// TIA Portal V16 program export: 7 tag tables, 0 data types, 4 data blocks, 31 code blocks (in call order from the OBs), 28 instance data blocks

VAR_GLOBAL   // PLC tag table "100固定地址变量表"
   ManAutoPB AT %I1.0 : Bool;   // 手动/自动   {ExternalVisible false}
   StartPB AT %I1.1 : Bool;   // 启动(固定)
   StopPB AT %I1.2 : Bool;   // 停止(固定)
   RestPB AT %I1.3 : Bool;   // 复位(固定)
   EM_PB AT %I1.4 : Bool;   // 急停(固定)
   Buzzer AT %Q0.4 : Bool;   // 蜂鸣器Bz
   R_LED AT %Q0.5 : Bool;   // 三色灯<红>
   G_LED AT %Q0.6 : Bool;   // 三色灯<绿>
   Y_LED AT %Q0.7 : Bool;   // 三色灯<黄>
   Auto_LED AT %Q1.0 : Bool;   // 自动灯
   Clock_Byte AT %MB0 : Byte;
   System_Byte AT %MB1 : Byte;
   "0.1s时钟" AT %M0.0 : Bool;
   "0.2s时钟" AT %M0.1 : Bool;
   "0.4s时钟" AT %M0.2 : Bool;
   "0.5s时钟" AT %M0.3 : Bool;
   "0.8s时钟" AT %M0.4 : Bool;
   "1.0s时钟" AT %M0.5 : Bool;
   "1.6s时钟" AT %M0.6 : Bool;
   "2s时钟" AT %M0.7 : Bool;
   初始 AT %M1.0 : Bool;
   DiagStatusUpdate AT %M1.1 : Bool;
   常ON AT %M1.2 : Bool;
   常OFF AT %M1.3 : Bool;
   Int_M AT %M2.0 : Bool;   // xx
   Init_2s AT %M2.1 : Bool;   // 初始2s
   Run_2s AT %M2.2 : Bool;   // 运行2s
   Run_3s AT %M2.3 : Bool;   // 运行3s
   Run_4s AT %M2.4 : Bool;   // 运行4s
   AutoStep_P AT %M2.6 : Bool;   // 单步脉冲
   Fault_Rest AT %M2.7 : Bool;   // 故障复位
   Com_EMO AT %M3.0 : Bool;   // 总急停
   Com_SLC AT %M3.1 : Bool;   // 总光栅
   Com_DSW AT %M3.2 : Bool;   // 总门SW
   Com_OtherSafe AT %M3.3 : Bool;   // 其它安全
   Com_AirALM AT %M3.4 : Bool;   // 总气压
   AllFaults AT %M6.0 : Bool;   // 全部故障
   AllALM AT %M6.1 : Bool;   // 严重报警
   AllERR AT %M6.2 : Bool;   // 错误报警
   AllPoint AT %M6.3 : Bool;   // 提示信息
   FaultBuzzer AT %M6.7 : Bool;   // 蜂鸣器
   ManMode AT %M100.0 : Bool;   // 手动(固定)
   InitPB_All AT %M105.0 : Bool;   // 全初始化
   SN1_InitPB AT %M110.0 : Bool;   // SN1初始化
   SN1_Initial AT %M110.3 : Bool;   // SN1初始位
   SN1_InitStart AT %M110.4 : Bool;   // SN1初始化开始
   SN1_InitEnd AT %M110.5 : Bool;   // SN1初始化结束
   SN2_InitPB AT %M112.0 : Bool;   // SN2初始化
   SN2_Initial AT %M112.3 : Bool;   // SN2初始位
   SN2_InitStart AT %M112.4 : Bool;   // SN2初始化开始
   SN2_InitEnd AT %M112.5 : Bool;   // SN2初始化结束
   SN3_InitPB AT %M114.0 : Bool;   // SN3初始化
   SN3_Initial AT %M114.3 : Bool;   // SN3初始位
   SN3_InitStart AT %M114.4 : Bool;   // SN3初始化开始
   SN3_InitEnd AT %M114.5 : Bool;   // SN3初始化结束
   SN4_InitPB AT %M116.0 : Bool;   // SN4初始化
   SN4_Initial AT %M116.3 : Bool;   // SN4初始位
   SN4_InitStart AT %M116.4 : Bool;   // SN4初始化开始
   SN4_InitEnd AT %M116.5 : Bool;   // SN4初始化结束
   SN5_InitPB AT %M118.0 : Bool;   // SN5初始化
   SN5_Initial AT %M118.3 : Bool;   // SN5初始位
   SN5_InitStart AT %M118.4 : Bool;   // SN5初始化开始
   SN5_InitEnd AT %M118.5 : Bool;   // SN5初始化结束
   SN6_InitPB AT %M120.0 : Bool;   // SN6初始化
   SN6_Initial AT %M120.3 : Bool;   // SN6初始位
   SN6_InitStart AT %M120.4 : Bool;   // SN6初始化开始
   SN6_InitEnd AT %M120.5 : Bool;   // SN6初始化结束
   SN7_InitPB AT %M122.0 : Bool;   // SN7初始化
   SN7_Initial AT %M122.3 : Bool;   // SN7初始位
   SN7_InitStart AT %M122.4 : Bool;   // SN7初始化开始
   SN7_InitEnd AT %M122.5 : Bool;   // SN7初始化结束
   SN8_InitPB AT %M124.0 : Bool;   // SN8初始化
   SN8_Initial AT %M124.3 : Bool;   // SN8初始位
   SN8_InitStart AT %M124.4 : Bool;   // SN8初始化开始
   SN8_InitEnd AT %M124.5 : Bool;   // SN8初始化结束
   SN9_InitPB AT %M126.0 : Bool;   // SN9初始化
   SN9_Initial AT %M126.3 : Bool;   // SN9初始位
   SN9_InitStart AT %M126.4 : Bool;   // SN9初始化开始
   SN9_InitEnd AT %M126.5 : Bool;   // SN9初始化结束
   SN10_InitPB AT %M128.0 : Bool;   // SN10初始化
   SN10_Initial AT %M128.3 : Bool;   // SN10初始位
   SN10_InitStart AT %M128.4 : Bool;   // SN10初始化开始
   SN10_InitEnd AT %M128.5 : Bool;   // SN10初始化结束
   SN11_InitPB AT %M130.0 : Bool;   // SN11初始化
   SN11_Initial AT %M130.3 : Bool;   // SN11初始位
   SN11_InitStart AT %M130.4 : Bool;   // SN11初始化开始
   SN11_InitEnd AT %M130.5 : Bool;   // SN11初始化结束
   SN12_InitPB AT %M132.0 : Bool;   // SN12初始化
   SN12_Initial AT %M132.3 : Bool;   // SN12初始位
   SN12_InitStart AT %M132.4 : Bool;   // SN12初始化开始
   SN12_InitEnd AT %M132.5 : Bool;   // SN12初始化结束
   SN13_InitPB AT %M134.0 : Bool;   // SN13初始化
   SN13_Initial AT %M134.3 : Bool;   // SN13初始位
   SN13_InitStart AT %M134.4 : Bool;   // SN13初始化开始
   SN13_InitEnd AT %M134.5 : Bool;   // SN13初始化结束
   SN14_InitPB AT %M136.0 : Bool;   // SN14初始化
   SN14_Initial AT %M136.3 : Bool;   // SN14初始位
   SN14_InitStart AT %M136.4 : Bool;   // SN14初始化开始
   SN14_InitEnd AT %M136.5 : Bool;   // SN14初始化结束
   SN15_InitPB AT %M138.0 : Bool;   // SN15初始化
   SN15_Initial AT %M138.3 : Bool;   // SN15初始位
   SN15_InitStart AT %M138.4 : Bool;   // SN15初始化开始
   SN15_InitEnd AT %M138.5 : Bool;   // SN15初始化结束
   SN16_InitPB AT %M140.0 : Bool;   // SN16初始化
   SN16_Initial AT %M140.3 : Bool;   // SN16初始位
   SN16_InitStart AT %M140.4 : Bool;   // SN16初始化开始
   SN16_InitEnd AT %M140.5 : Bool;   // SN16初始化结束
   SN17_InitPB AT %M142.0 : Bool;   // SN17初始化
   SN17_Initial AT %M142.3 : Bool;   // SN17初始位
   SN17_InitStart AT %M142.4 : Bool;   // SN17初始化开始
   SN17_InitEnd AT %M142.5 : Bool;   // SN17初始化结束
   SN18_InitPB AT %M144.0 : Bool;   // SN18初始化
   SN18_Initial AT %M144.3 : Bool;   // SN18初始位
   SN18_InitStart AT %M144.4 : Bool;   // SN18初始化开始
   SN18_InitEnd AT %M144.5 : Bool;   // SN18初始化结束
   SN19_InitPB AT %M146.0 : Bool;   // SN19初始化
   SN19_Initial AT %M146.3 : Bool;   // SN19初始位
   SN19_InitStart AT %M146.4 : Bool;   // SN19初始化开始
   SN19_InitEnd AT %M146.5 : Bool;   // SN19初始化结束
   SN20_InitPB AT %M148.0 : Bool;   // SN20初始化
   SN20_Initial AT %M148.3 : Bool;   // SN20初始位
   SN20_InitStart AT %M148.4 : Bool;   // SN20初始化开始
   SN20_InitEnd AT %M148.5 : Bool;   // SN20初始化结束
   AutoMode AT %M150.0 : Bool;   // 自动模式
   AutoCont_Cut AT %M150.1 : Bool;   // 自动条件
   AutoPB_OFF AT %M150.2 : Bool;   // 自动OFF
   AutoStopReq AT %M150.3 : Bool;   // 自动停止要求
   Auto AT %M150.4 : Bool;   // 自动中
   InitPos AT %M150.5 : Bool;   // 初始位置
   AutoStop AT %M150.6 : Bool;   // 自动停止
   AlarmStop AT %M151.0 : Bool;   // 故障停止
   ErrorStop AT %M151.1 : Bool;   // 错误停止
   "SN1_Step(入口)" AT %MW200 : Int;   // SN1流程步
   "SN1_Start(入口)" AT %M250.0 : Bool;   // SN1开始
   "SN1_End(入口)" AT %M250.1 : Bool;   // SN1结束
   "SN1_搬入(入口)" AT %M250.2 : Bool;
   "SN1_搬出(入口)" AT %M250.3 : Bool;
   "SN2_Step(出口)" AT %MW202 : Int;   // SN2流程步
   "SN2_Start(出口)" AT %M252.0 : Bool;   // SN2开始
   "SN2_End(出口)" AT %M252.1 : Bool;   // SN2结束
   "SN2_搬入(出口)" AT %M252.2 : Bool;
   "SN2_搬出(出口)" AT %M252.3 : Bool;
   "SN3_Step(ST01上)" AT %MW204 : Int;   // SN3流程步
   "SN3_Start(ST01上)" AT %M254.0 : Bool;   // SN3开始
   "SN3_End(ST01上)" AT %M254.1 : Bool;   // SN3结束
   "SN3_搬入(ST01上)" AT %M254.2 : Bool;
   "SN3_搬出(ST01上)" AT %M254.3 : Bool;
   ST01放行标志 AT %M254.7 : Bool;
   "SN4_Step(ST02上)" AT %MW206 : Int;   // SN4流程步
   "SN4_Start(ST02上)" AT %M256.0 : Bool;   // SN4开始
   "SN4_End(ST02上)" AT %M256.1 : Bool;   // SN4结束
   "SN4_搬入(ST02上)" AT %M256.2 : Bool;
   "SN4_搬出(ST02上)" AT %M256.3 : Bool;
   ST02放行标志 AT %M256.7 : Bool;
   "SN5_Step(ST03上)" AT %MW208 : Int;   // SN5流程步
   "SN5_Start(ST03上)" AT %M258.0 : Bool;   // SN5开始
   "SN5_End(ST03上)" AT %M258.1 : Bool;   // SN5结束
   "SN5_搬入(ST03上)" AT %M258.2 : Bool;
   "SN5_搬出(ST03上)" AT %M258.3 : Bool;
   ST03放行标志 AT %M258.7 : Bool;
   "SN6_Step(ST04上)" AT %MW214 : Int;   // SN6流程步
   "SN6_Start(ST04上)" AT %M260.0 : Bool;   // SN6开始
   "SN6_End(ST04上)" AT %M260.1 : Bool;   // SN6结束
   "SN6_搬入(ST04上)" AT %M260.2 : Bool;
   "SN6_搬出(ST04上)" AT %M260.3 : Bool;
   ST04放行标志 AT %M260.7 : Bool;
   "SN7_Step(ST05上)" AT %MW216 : Int;   // SN7流程步
   "SN7_Start(ST05上)" AT %M262.0 : Bool;   // SN7开始
   "SN7_End(ST05上)" AT %M262.1 : Bool;   // SN7结束
   "SN7_搬入(ST05上)" AT %M262.2 : Bool;
   "SN7_搬出(ST05上)" AT %M262.3 : Bool;
   ST05放行标志 AT %M262.7 : Bool;
   "SN8_Step(ST06上)" AT %MW218 : Int;   // SN8流程步
   "SN8_Start(ST06上)" AT %M264.0 : Bool;   // SN8开始
   "SN8_End(ST06上)" AT %M264.1 : Bool;   // SN8结束
   "SN8_搬入(ST06上)" AT %M264.2 : Bool;
   "SN8_搬出(ST06上)" AT %M264.3 : Bool;
   ST06放行标志 AT %M264.7 : Bool;
   "SN9_Step(ST07上)" AT %MW222 : Int;   // SN9流程步
   "SN9_Start(ST07上)" AT %M265.0 : Bool;   // SN9开始
   "SN9_End(ST07上)" AT %M266.1 : Bool;   // SN9结束
   "SN9_搬入(ST07上)" AT %M266.2 : Bool;
   "SN9_搬出(ST07上)" AT %M266.3 : Bool;
   ST07放行标志 AT %M266.7 : Bool;
   "SN10_Step(ST08上)" AT %MW224 : Int;   // SN10流程步
   "SN10_Start(ST08上)" AT %M268.0 : Bool;   // SN10开始
   "SN10_End(ST08上)" AT %M268.1 : Bool;   // SN10结束
   "SN10_搬入(ST08上)" AT %M268.2 : Bool;
   "SN10_搬出(ST08上)" AT %M268.3 : Bool;
   ST08放行标志 AT %M268.7 : Bool;
   "SN11_Step(ST09上)" AT %MW226 : Int;   // SN11流程步
   "SN11_Start(ST09上)" AT %M270.0 : Bool;   // SN11开始
   "SN11_End(ST09上)" AT %M270.1 : Bool;   // SN11结束
   "SN11_搬入(ST09上)" AT %M270.2 : Bool;
   "SN11_搬出(ST09上)" AT %M270.3 : Bool;
   ST09放行标志 AT %M270.7 : Bool;
   "SN12_Step(ST10上)" AT %MW228 : Int;   // SN12流程步
   "SN12_Start(ST10上)" AT %M272.0 : Bool;   // SN12开始
   "SN12_End(ST10上)" AT %M272.1 : Bool;   // SN12结束
   "SN12_搬入(ST10上)" AT %M272.2 : Bool;
   "SN12_搬出(ST10上)" AT %M272.3 : Bool;
   ST10放行标志 AT %M272.7 : Bool;
   "SN13_Step(ST11上)" AT %MW230 : Int;   // SN13流程步
   "SN13_Start(ST11上)" AT %M274.0 : Bool;   // SN13开始
   "SN13_End(ST11上)" AT %M274.1 : Bool;   // SN13结束
   "SN13_搬入(ST11上)" AT %M274.2 : Bool;
   "SN13_搬出(ST11上)" AT %M274.3 : Bool;
   ST11放行标志 AT %M274.7 : Bool;
   "SN14_Step(ST12上)" AT %MW232 : Int;   // SN14流程步
   "SN14_Start(ST12上)" AT %M276.0 : Bool;   // SN14开始
   "SN14_End(ST12上)" AT %M276.1 : Bool;   // SN14结束
   "SN14_搬入(ST12上)" AT %M276.2 : Bool;
   "SN14_搬出(ST12上)" AT %M276.3 : Bool;
   ST12放行标志 AT %M276.7 : Bool;
   "SN15_Step(ST03下)" AT %MW234 : Int;   // SN15流程步
   SN15_Start AT %M278.0 : Bool;   // SN15开始
   SN15_End AT %M278.1 : Bool;   // SN15结束
   SN15_搬入 AT %M278.2 : Bool;
   SN15_搬出 AT %M278.3 : Bool;
   "SN16_Step(ST02下)" AT %MW236 : Int;   // SN16流程步
   SN16_Start AT %M280.0 : Bool;   // SN16开始
   SN16_End AT %M280.1 : Bool;   // SN16结束
   SN16_搬入 AT %M280.2 : Bool;
   SN16_搬出 AT %M280.3 : Bool;
   "SN17_Step(ST01下)" AT %MW238 : Int;   // SN17流程步
   SN17_Start AT %M282.0 : Bool;   // SN17开始
   SN17_End AT %M282.1 : Bool;   // SN17结束
   SN17_搬入 AT %M282.2 : Bool;
   SN17_搬出 AT %M282.3 : Bool;
   SN18_Step AT %MW240 : Int;   // SN18流程步
   SN18_Start AT %M284.0 : Bool;   // SN18开始
   SN18_End AT %M284.1 : Bool;   // SN18结束
   SN18_搬入 AT %M284.2 : Bool;
   SN18_搬出 AT %M284.3 : Bool;
   SN19_Step AT %MW242 : Int;   // SN19流程步
   SN19_Start AT %M286.0 : Bool;   // SN19开始
   SN19_End AT %M286.1 : Bool;   // SN19结束
   SN19_搬入 AT %M286.2 : Bool;
   SN19_搬出 AT %M286.3 : Bool;
   SN20_Step AT %MW244 : Int;   // SN20流程步
   SN20_Start AT %M288.0 : Bool;   // SN20开始
   SN20_End AT %M288.1 : Bool;   // SN20结束
   SN20_搬入 AT %M288.2 : Bool;
   SN20_搬出 AT %M288.3 : Bool;
   AutoStep AT %M600.0 : Bool;   // 自动单步
   LampTest AT %M600.1 : Bool;   // 灯测试
   Durable AT %M600.2 : Bool;   // 耐久模式
   ST01屏蔽 AT %M650.0 : Bool;
   ST02屏蔽 AT %M650.1 : Bool;
   ST03屏蔽 AT %M650.2 : Bool;
   ST04屏蔽 AT %M650.3 : Bool;
   ST05屏蔽 AT %M650.4 : Bool;
   ST06屏蔽 AT %M650.5 : Bool;
   ST07屏蔽 AT %M650.6 : Bool;
   ST08屏蔽 AT %M650.7 : Bool;
   ST09屏蔽 AT %M651.0 : Bool;
   ST10屏蔽 AT %M651.1 : Bool;
   ST11屏蔽 AT %M651.2 : Bool;
   ST12屏蔽 AT %M651.3 : Bool;
   ST13屏蔽 AT %M651.4 : Bool;
   ST14屏蔽 AT %M651.5 : Bool;
   ST15屏蔽 AT %M651.6 : Bool;
   ST16屏蔽 AT %M651.7 : Bool;
   ST17屏蔽 AT %M652.0 : Bool;
   ST18屏蔽 AT %M652.1 : Bool;
   ST19屏蔽 AT %M652.2 : Bool;
   ST20屏蔽 AT %M652.3 : Bool;
   生产数量清零 AT %M695.0 : Bool;
   累计数量清零 AT %M695.1 : Bool;
END_VAR

VAR_GLOBAL   // PLC tag table "101生产数据变量表"
   当前日期年 AT %MW700 : Int;
   当前日期月 AT %MW702 : Int;
   当前日期日 AT %MW704 : Int;
   当前日期时 AT %MW706 : Int;
   当前日期分 AT %MW708 : Int;
   当前日期秒 AT %MW710 : Int;
   开机日期年 AT %MW720 : Int;
   开机日期月 AT %MW722 : Int;
   开机日期日 AT %MW724 : Int;
   开机日期时 AT %MW726 : Int;
   开机日期分 AT %MW728 : Int;
   开机日期秒 AT %MW730 : Int;
   "运行时间(H)" AT %MW740 : Int;
   "运行时间(M)" AT %MW742 : Int;
   "停止时间(H)" AT %MW744 : Int;
   "停止时间(M)" AT %MW746 : Int;
   "故障时间(H)" AT %MW748 : Int;
   "故障时间(M)" AT %MW750 : Int;
   生产数量 AT %MD760 : DInt;
   OK数量 AT %MD764 : DInt;
   NG数量 AT %MD768 : DInt;
   累计数量 AT %MD772 : DInt;
   实时节拍 AT %MW780 : Int;
   工作节拍 AT %MW782 : Int;
   "开机时间(H)" AT %MW732 : Int;
   "开机时间(M)" AT %MW734 : Int;
   "稼动率%" AT %MW752 : Int;
   "合格率%" AT %MW776 : Int;
   PPM AT %MW778 : Int;
   设置日期年 AT %MW800 : Int;
   设置日期月 AT %MW802 : Int;
   设置日期日 AT %MW804 : Int;
   设置日期时 AT %MW806 : Int;
   设置日期分 AT %MW808 : Int;
   设置日期秒 AT %MW810 : Int;
   日期设置通知 AT %M812.0 : Bool;
END_VAR

VAR_GLOBAL   // PLC tag table "102故障数据变量表"
   HMI总急停报警 AT %MW6000 : Int;
   HMI总光栅报警 AT %MW6002 : Int;
   HMI总安全门报警 AT %MW6004 : Int;
   HMI总其它安全报警 AT %MW6006 : Int;
   HMI总气压报警 AT %MW6008 : Int;
   HMI总滚筒故障1 AT %MW6010 : Int;
   HMI总滚筒故障2 AT %MW6012 : Int;
   HMI总滚筒故障3 AT %MW6014 : Int;
   HMI总滚筒超时1 AT %MW6016 : Int;
   HMI总滚筒超时2 AT %MW6018 : Int;
   HMI总滚筒超时3 AT %MW6020 : Int;
   HMI总变频器故障 AT %MW6022 : Int;
   HMI总变频器未运行故障 AT %MW6024 : Int;
   HMI总变频器过载故障 AT %MW6026 : Int;
   HMI总变频器超时故障 AT %MW6028 : Int;
   HMI阀出动作超时1 AT %MW6030 : Int;
   HMI阀出动作超时2 AT %MW6032 : Int;
   HMI阀出动作超时3 AT %MW6034 : Int;
   HMI阀出动作超时4 AT %MW6036 : Int;
   HMI阀出动作超时5 AT %MW6038 : Int;
   HMI阀回动作超时1 AT %MW6040 : Int;
   HMI阀回动作超时2 AT %MW6042 : Int;
   HMI阀回动作超时3 AT %MW6044 : Int;
   HMI阀回动作超时4 AT %MW6046 : Int;
   HMI阀回动作超时5 AT %MW6048 : Int;
   HMI阀传感器全到位故障1 AT %MW6050 : Int;
   HMI阀传感器全到位故障2 AT %MW6052 : Int;
   HMI阀传感器全到位故障3 AT %MW6054 : Int;
   HMI阀传感器全到位故障4 AT %MW6056 : Int;
   HMI阀传感器全到位故障5 AT %MW6058 : Int;
   HMI阀传感器交叉ON故障1 AT %MW6060 : Int;
   HMI阀传感器交叉ON故障2 AT %MW6062 : Int;
   HMI阀传感器交叉ON故障3 AT %MW6064 : Int;
   HMI阀传感器交叉ON故障4 AT %MW6066 : Int;
   HMI阀传感器交叉ON故障5 AT %MW6068 : Int;
   HMI伺服报警 AT %MW6070 : Int;
   HMI伺服故障 AT %MW6072 : Int;
   HMI伺服未准备好 AT %MW6074 : Int;
   HMI伺服未回零故障 AT %MW6076 : Int;
   HMI伺服未运行故障 AT %MW6078 : Int;
   HM伺服正极限故障 AT %MW6080 : Int;
   HMI伺服负极限故障 AT %MW6082 : Int;
   HMI视觉故障 AT %MW6084 : Int;
   HMI机器人故障 AT %MW6086 : Int;
   HMI通信故障 AT %MW6088 : Int;
   HMI模拟量上极限故障 AT %MW6090 : Int;
   HMI模拟量下极限故障 AT %MW6092 : Int;
   HMI其它类故障 AT %MW6094 : Int;
   HMI传感器故障1 AT %MW6096 : Int;
   HMI传感器故障2 AT %MW6098 : Int;
   HMI传感器故障3 AT %MW6100 : Int;
   HMI传感器故障4 AT %MW6102 : Int;
   HMI传感器故障5 AT %MW6104 : Int;
   HMI传感器故障6 AT %MW6106 : Int;
   HMI动作异常1 AT %MW6108 : Int;
   HMI动作异常2 AT %MW6110 : Int;
   HMI动作异常3 AT %MW6112 : Int;
END_VAR

VAR_GLOBAL   // PLC tag table "103输入点变量表"
   EN_INV1故障 AT %I2.0 : Bool;
   Air故障 AT %I2.1 : Bool;
   EN_前端LS AT %I2.2 : Bool;
   EN_后端LS AT %I2.3 : Bool;
   EN_阻挡上升端 AT %I2.4 : Bool;
   EN_阻挡下降端 AT %I2.5 : Bool;
   EN_上升端 AT %I2.6 : Bool;
   EN_下降端 AT %I2.7 : Bool;
   EX_INV2故障 AT %I3.0 : Bool;
   干涉确认LS AT %I3.1 : Bool;
   EX_前端LS AT %I3.2 : Bool;
   EX_后端LS AT %I3.3 : Bool;
   EX_阻挡上升端 AT %I3.4 : Bool;
   EX_阻挡下降端 AT %I3.5 : Bool;
   EX_上升端 AT %I3.6 : Bool;
   EX_下降端 AT %I3.7 : Bool;
   ST01上层前端LS AT %I4.0 : Bool;
   ST01上层后端LS AT %I4.1 : Bool;
   ST01上阻挡上升端 AT %I4.2 : Bool;
   ST01上阻挡下降端 AT %I4.3 : Bool;
   ST01下层前端LS AT %I4.4 : Bool;
   ST01下层后端LS AT %I4.5 : Bool;
   ST01下阻挡上升端 AT %I4.6 : Bool;
   ST01下阻挡下降端 AT %I4.7 : Bool;
   ST02上层前端LS AT %I5.0 : Bool;
   ST02上层后端LS AT %I5.1 : Bool;
   ST02上阻挡上升端 AT %I5.2 : Bool;
   ST02上阻挡下降端 AT %I5.3 : Bool;
   ST02下层前端LS AT %I5.4 : Bool;
   ST02下层后端LS AT %I5.5 : Bool;
   ST02下阻挡上升端 AT %I5.6 : Bool;
   ST02下阻挡下降端 AT %I5.7 : Bool;
   ST03上层前端LS AT %I6.0 : Bool;
   ST03上层后端LS AT %I6.1 : Bool;
   ST03上阻挡上升端 AT %I6.2 : Bool;
   ST03上阻挡下降端 AT %I6.3 : Bool;
   ST03下层前端LS AT %I6.4 : Bool;
   ST03下层后端LS AT %I6.5 : Bool;
   ST03下阻挡上升端 AT %I6.6 : Bool;
   ST03下阻挡下降端 AT %I6.7 : Bool;
   ST04上层前端LS AT %I7.0 : Bool;
   ST04上层后端LS AT %I7.1 : Bool;
   ST04上阻挡上升端 AT %I7.2 : Bool;
   ST04上阻挡下降端 AT %I7.3 : Bool;
   ST05上层前端LS AT %I7.4 : Bool;
   ST05上层后端LS AT %I7.5 : Bool;
   ST05上阻挡上升端 AT %I7.6 : Bool;
   ST05上阻挡下降端 AT %I7.7 : Bool;
   前段_INV3故障 AT %I8.0 : Bool;
   前段_INV4故障 AT %I8.1 : Bool;
   后段_INV5故障 AT %I8.2 : Bool;
   后段_INV6故障 AT %I8.3 : Bool;
   ST06上层前端LS AT %I8.4 : Bool;
   ST06上层后端LS AT %I8.5 : Bool;
   ST06上阻挡上升端 AT %I8.6 : Bool;
   ST06上阻挡下降端 AT %I8.7 : Bool;
   ST07上层前端LS AT %I9.0 : Bool;
   ST07上层后端LS AT %I9.1 : Bool;
   ST07上阻挡上升端 AT %I9.2 : Bool;
   ST07上阻挡下降端 AT %I9.3 : Bool;
   ST08上层前端LS AT %I9.4 : Bool;
   ST08上层后端LS AT %I9.5 : Bool;
   ST08上阻挡上升端 AT %I9.6 : Bool;
   ST08上阻挡下降端 AT %I9.7 : Bool;
   ST09上层前端LS AT %I10.0 : Bool;
   ST09上层后端LS AT %I10.1 : Bool;
   ST09上阻挡上升端 AT %I10.2 : Bool;
   ST09上阻挡下降端 AT %I10.3 : Bool;
   ST10上层前端LS AT %I10.4 : Bool;
   ST10上层后端LS AT %I10.5 : Bool;
   ST10上阻挡上升端 AT %I10.6 : Bool;
   ST10上阻挡下降端 AT %I10.7 : Bool;
   ST11上层前端LS AT %I11.0 : Bool;
   ST11上层后端LS AT %I11.1 : Bool;
   ST11上阻挡上升端 AT %I11.2 : Bool;
   ST11上阻挡下降端 AT %I11.3 : Bool;
   ST12上层前端LS AT %I11.4 : Bool;
   ST12上层后端LS AT %I11.5 : Bool;
   ST12上阻挡上升端 AT %I11.6 : Bool;
   ST12上阻挡下降端 AT %I11.7 : Bool;
   ST01急停EM AT %I12.0 : Bool;
   ST01放行SB AT %I12.1 : Bool;
   ST02急停EM AT %I12.2 : Bool;
   ST02放行SB AT %I12.3 : Bool;
   ST03急停EM AT %I12.4 : Bool;
   ST03放行SB AT %I12.5 : Bool;
   ST04急停EM AT %I12.6 : Bool;
   ST04放行SB AT %I12.7 : Bool;
   ST05急停EM AT %I13.0 : Bool;
   ST05放行SB AT %I13.1 : Bool;
   ST06急停EM AT %I13.2 : Bool;
   ST06放行SB AT %I13.3 : Bool;
   ST07急停EM AT %I14.0 : Bool;
   ST07放行SB AT %I14.1 : Bool;
   ST08急停EM AT %I14.2 : Bool;
   ST08放行SB AT %I14.3 : Bool;
   ST09急停EM AT %I14.4 : Bool;
   ST09放行SB AT %I14.5 : Bool;
   ST10急停EM AT %I14.6 : Bool;
   ST10放行SB AT %I14.7 : Bool;
   ST11急停EM AT %I15.0 : Bool;
   ST11放行SB AT %I15.1 : Bool;
   ST12急停EM AT %I15.2 : Bool;
   ST12放行SB AT %I15.3 : Bool;
END_VAR

VAR_GLOBAL   // PLC tag table "104输出点变量表"
   EN_INV1正转 AT %Q2.0 : Bool;
   EN_INV1反转 AT %Q2.1 : Bool;
   EN_INV1速度 AT %Q2.2 : Bool;
   EN_INV1复位 AT %Q2.3 : Bool;
   EN_阻挡下降 AT %Q2.5 : Bool;
   EN_提升机上升 AT %Q2.6 : Bool;
   EN_提升机下降 AT %Q2.7 : Bool;
   EX_INV2正转 AT %Q3.0 : Bool;
   EX_INV2反转 AT %Q3.1 : Bool;
   EX_INV2速度 AT %Q3.2 : Bool;
   EX_INV2复位 AT %Q3.3 : Bool;
   EX_阻挡下降 AT %Q3.5 : Bool;
   EX_提升机上升 AT %Q3.6 : Bool;
   EX_提升机下降 AT %Q3.7 : Bool;
   ST01上阻挡下降 AT %Q4.1 : Bool;
   ST01下阻挡下降 AT %Q4.3 : Bool;
   ST02上阻挡下降 AT %Q4.5 : Bool;
   ST02下阻挡下降 AT %Q4.7 : Bool;
   ST03上阻挡下降 AT %Q5.1 : Bool;
   ST03下阻挡下降 AT %Q5.3 : Bool;
   ST04上阻挡下降 AT %Q5.5 : Bool;
   ST05上阻挡下降 AT %Q5.7 : Bool;
   前段_INV3正转 AT %Q8.0 : Bool;
   前段_INV3速度1 AT %Q8.1 : Bool;
   前段_INV3速度2 AT %Q8.2 : Bool;
   前段_INV3复位 AT %Q8.3 : Bool;
   前段_INV4正转 AT %Q8.4 : Bool;
   前段_INV4速度1 AT %Q8.5 : Bool;
   前段_INV4速度2 AT %Q8.6 : Bool;
   前段_INV4复位 AT %Q8.7 : Bool;
   后段_INV5正转 AT %Q9.0 : Bool;
   后段_INV5速度1 AT %Q9.1 : Bool;
   后段_INV5速度2 AT %Q9.2 : Bool;
   后段_INV5复位 AT %Q9.3 : Bool;
   后段_INV6正转 AT %Q9.4 : Bool;
   后段_INV6速度1 AT %Q9.5 : Bool;
   后段_INV6速度2 AT %Q9.6 : Bool;
   后段_INV6复位 AT %Q9.7 : Bool;
   ST06上阻挡下降 AT %Q10.1 : Bool;
   ST07上阻挡下降 AT %Q10.3 : Bool;
   ST08上阻挡下降 AT %Q10.5 : Bool;
   ST09上阻挡下降 AT %Q11.1 : Bool;
   ST10上阻挡下降 AT %Q11.3 : Bool;
   ST11上阻挡下降 AT %Q11.5 : Bool;
   ST12上阻挡下降 AT %Q11.7 : Bool;
   ST01放行LED AT %Q12.0 : Bool;
   ST02放行LED AT %Q12.1 : Bool;
   ST03放行LED AT %Q12.2 : Bool;
   ST04放行LED AT %Q12.3 : Bool;
   ST05放行LED AT %Q12.4 : Bool;
   ST06放行LED AT %Q12.5 : Bool;
   ST07放行LED AT %Q13.0 : Bool;
   ST08放行LED AT %Q13.1 : Bool;
   ST09放行LED AT %Q13.2 : Bool;
   ST10放行LED AT %Q13.3 : Bool;
   ST11放行LED AT %Q13.4 : Bool;
   ST12放行LED AT %Q13.5 : Bool;
END_VAR

VAR_GLOBAL   // PLC tag table "105阀控制变量表"
   EN_阻挡下指令自动 AT %M2000.0 : Bool;
   EN_阻挡上指令自动 AT %M2000.1 : Bool;
   EN_提升机下指令自动 AT %M2000.4 : Bool;
   EN_提升机上指令自动 AT %M2000.5 : Bool;
   EX_阻挡下指令自动 AT %M2001.0 : Bool;
   EX_阻挡上指令自动 AT %M2001.1 : Bool;
   EX_提升机下指令自动 AT %M2001.4 : Bool;
   EX_提升机上指令自动 AT %M2001.5 : Bool;
   ST01上阻挡下指令自动 AT %M2002.0 : Bool;
   ST01上阻挡上指令自动 AT %M2002.1 : Bool;
   ST01下阻挡下指令自动 AT %M2002.4 : Bool;
   ST01下阻挡上指令自动 AT %M2002.5 : Bool;
   ST02上阻挡下指令自动 AT %M2003.0 : Bool;
   ST02上阻挡上指令自动 AT %M2003.1 : Bool;
   ST02下阻挡下指令自动 AT %M2003.4 : Bool;
   ST02下阻挡上指令自动 AT %M2003.5 : Bool;
   ST03上阻挡下指令自动 AT %M2004.0 : Bool;
   ST03上阻挡上指令自动 AT %M2004.1 : Bool;
   ST03下阻挡下指令自动 AT %M2004.4 : Bool;
   ST03下阻挡上指令自动 AT %M2004.5 : Bool;
   ST04上阻挡下指令自动 AT %M2005.0 : Bool;
   ST04上阻挡上指令自动 AT %M2005.1 : Bool;
   ST05上阻挡下指令自动 AT %M2005.4 : Bool;
   ST05上阻挡上指令自动 AT %M2005.5 : Bool;
   ST06上阻挡下指令自动 AT %M2006.0 : Bool;
   ST06上阻挡上指令自动 AT %M2006.1 : Bool;
   ST07上阻挡下指令自动 AT %M2006.4 : Bool;
   ST07上阻挡上指令自动 AT %M2006.5 : Bool;
   ST08上阻挡下指令自动 AT %M2007.0 : Bool;
   ST08上阻挡上指令自动 AT %M2007.1 : Bool;
   ST09上阻挡下指令自动 AT %M2007.4 : Bool;
   ST09上阻挡上指令自动 AT %M2007.5 : Bool;
   ST10上阻挡下指令自动 AT %M2008.0 : Bool;
   ST10上阻挡上指令自动 AT %M2008.1 : Bool;
   ST11上阻挡下指令自动 AT %M2008.4 : Bool;
   ST11上阻挡上指令自动 AT %M2008.5 : Bool;
   ST12上阻挡下指令自动 AT %M2009.0 : Bool;
   ST12上阻挡上指令自动 AT %M2009.1 : Bool;
   阀20进指令自动 AT %M2009.4 : Bool;
   阀20回指令自动 AT %M2009.5 : Bool;
   阀21进指令自动 AT %M2010.0 : Bool;
   阀21回指令自动 AT %M2010.1 : Bool;
   阀22进指令自动 AT %M2010.4 : Bool;
   阀22回指令自动 AT %M2010.5 : Bool;
   阀23进指令自动 AT %M2011.0 : Bool;
   阀23回指令自动 AT %M2011.1 : Bool;
   阀24进指令自动 AT %M2011.4 : Bool;
   阀24回指令自动 AT %M2011.5 : Bool;
   阀25进指令自动 AT %M2012.0 : Bool;
   阀25回指令自动 AT %M2012.1 : Bool;
   阀26进指令自动 AT %M2012.4 : Bool;
   阀26回指令自动 AT %M2012.5 : Bool;
   阀27进指令自动 AT %M2013.0 : Bool;
   阀27回指令自动 AT %M2013.1 : Bool;
   阀28进指令自动 AT %M2013.4 : Bool;
   阀28回指令自动 AT %M2013.5 : Bool;
   阀29进指令自动 AT %M2014.0 : Bool;
   阀29回指令自动 AT %M2014.1 : Bool;
   阀30进指令自动 AT %M2014.4 : Bool;
   阀30回指令自动 AT %M2014.5 : Bool;
   阀31进指令自动 AT %M2015.0 : Bool;
   阀31回指令自动 AT %M2015.1 : Bool;
   阀32进指令自动 AT %M2015.4 : Bool;
   阀32回指令自动 AT %M2015.5 : Bool;
   阀33进指令自动 AT %M2016.0 : Bool;
   阀33回指令自动 AT %M2016.1 : Bool;
   阀34进指令自动 AT %M2016.4 : Bool;
   阀34回指令自动 AT %M2016.5 : Bool;
   阀35进指令自动 AT %M2017.0 : Bool;
   阀35回指令自动 AT %M2017.1 : Bool;
   阀36进指令自动 AT %M2017.4 : Bool;
   阀36回指令自动 AT %M2017.5 : Bool;
   阀37进指令自动 AT %M2018.0 : Bool;
   阀37回指令自动 AT %M2018.1 : Bool;
   阀38进指令自动 AT %M2018.4 : Bool;
   阀38回指令自动 AT %M2018.5 : Bool;
   阀39进指令自动 AT %M2019.0 : Bool;
   阀39回指令自动 AT %M2019.1 : Bool;
   阀40进指令自动 AT %M2019.4 : Bool;
   阀40回指令自动 AT %M2019.5 : Bool;
   阀41进指令自动 AT %M2020.0 : Bool;
   阀41回指令自动 AT %M2020.1 : Bool;
   阀42进指令自动 AT %M2020.4 : Bool;
   阀42回指令自动 AT %M2020.5 : Bool;
   阀43进指令自动 AT %M2021.0 : Bool;
   阀43回指令自动 AT %M2021.1 : Bool;
   阀44进指令自动 AT %M2021.4 : Bool;
   阀44回指令自动 AT %M2021.5 : Bool;
   阀45进指令自动 AT %M2022.0 : Bool;
   阀45回指令自动 AT %M2022.1 : Bool;
   阀46进指令自动 AT %M2022.4 : Bool;
   阀46回指令自动 AT %M2022.5 : Bool;
   阀47进指令自动 AT %M2023.0 : Bool;
   阀47回指令自动 AT %M2023.1 : Bool;
   阀48进指令自动 AT %M2023.4 : Bool;
   阀48回指令自动 AT %M2023.5 : Bool;
   EN_阻挡下指令手动 AT %M1000.0 : Bool;
   EN_阻挡上指令手动 AT %M1000.1 : Bool;
   EN_提升机下指令手动 AT %M1000.4 : Bool;
   EN_提升机上指令手动 AT %M1000.5 : Bool;
   EX_阻挡下指令手动 AT %M1001.0 : Bool;
   EX_阻挡上指令手动 AT %M1001.1 : Bool;
   EX_提升机下指令手动 AT %M1001.4 : Bool;
   EX_提升机上指令手动 AT %M1001.5 : Bool;
   ST01上阻挡下指令手动 AT %M1002.0 : Bool;
   ST01上阻挡上指令手动 AT %M1002.1 : Bool;
   ST01下阻挡下指令手动 AT %M1002.4 : Bool;
   ST01下阻挡上指令手动 AT %M1002.5 : Bool;
   ST02上阻挡下指令手动 AT %M1003.0 : Bool;
   ST02上阻挡上指令手动 AT %M1003.1 : Bool;
   ST02下阻挡下指令手动 AT %M1003.4 : Bool;
   ST02下阻挡上指令手动 AT %M1003.5 : Bool;
   ST03上阻挡下指令手动 AT %M1004.0 : Bool;
   ST03上阻挡上指令手动 AT %M1004.1 : Bool;
   ST03下阻挡下指令手动 AT %M1004.4 : Bool;
   ST03下阻挡上指令手动 AT %M1004.5 : Bool;
   ST04上阻挡下指令手动 AT %M1005.0 : Bool;
   ST04上阻挡上指令手动 AT %M1005.1 : Bool;
   ST05上阻挡下指令手动 AT %M1005.4 : Bool;
   ST05上阻挡上指令手动 AT %M1005.5 : Bool;
   ST06上阻挡下指令手动 AT %M1006.0 : Bool;
   ST06上阻挡上指令手动 AT %M1006.1 : Bool;
   ST07上阻挡下指令手动 AT %M1006.4 : Bool;
   ST07上阻挡上指令手动 AT %M1006.5 : Bool;
   ST08上阻挡下指令手动 AT %M1007.0 : Bool;
   ST08上阻挡上指令手动 AT %M1007.1 : Bool;
   ST09上阻挡下指令手动 AT %M1007.4 : Bool;
   ST09上阻挡上指令手动 AT %M1007.5 : Bool;
   ST10上阻挡下指令手动 AT %M1008.0 : Bool;
   ST10上阻挡上指令手动 AT %M1008.1 : Bool;
   ST11上阻挡下指令手动 AT %M1008.4 : Bool;
   ST11上阻挡上指令手动 AT %M1008.5 : Bool;
   ST12上阻挡下指令手动 AT %M1009.0 : Bool;
   ST12上阻挡上指令手动 AT %M1009.1 : Bool;
   阀20进指令手动 AT %M1009.4 : Bool;
   阀20回指令手动 AT %M1009.5 : Bool;
   阀21进指令手动 AT %M1010.0 : Bool;
   阀21回指令手动 AT %M1010.1 : Bool;
   阀22进指令手动 AT %M1010.4 : Bool;
   阀22回指令手动 AT %M1010.5 : Bool;
   阀23进指令手动 AT %M1011.0 : Bool;
   阀23回指令手动 AT %M1011.1 : Bool;
   阀24进指令手动 AT %M1011.4 : Bool;
   阀24回指令手动 AT %M1011.5 : Bool;
   阀25进指令手动 AT %M1012.0 : Bool;
   阀25回指令手动 AT %M1012.1 : Bool;
   阀26进指令手动 AT %M1012.4 : Bool;
   阀26回指令手动 AT %M1012.5 : Bool;
   阀27进指令手动 AT %M1013.0 : Bool;
   阀27回指令手动 AT %M1013.1 : Bool;
   阀28进指令手动 AT %M1013.4 : Bool;
   阀28回指令手动 AT %M1013.5 : Bool;
   阀29进指令手动 AT %M1014.0 : Bool;
   阀29回指令手动 AT %M1014.1 : Bool;
   阀30进指令手动 AT %M1014.4 : Bool;
   阀30回指令手动 AT %M1014.5 : Bool;
   阀31进指令手动 AT %M1015.0 : Bool;
   阀31回指令手动 AT %M1015.1 : Bool;
   阀32进指令手动 AT %M1015.4 : Bool;
   阀32回指令手动 AT %M1015.5 : Bool;
   阀33进指令手动 AT %M1016.0 : Bool;
   阀33回指令手动 AT %M1016.1 : Bool;
   阀34进指令手动 AT %M1016.4 : Bool;
   阀34回指令手动 AT %M1016.5 : Bool;
   阀35进指令手动 AT %M1017.0 : Bool;
   阀35回指令手动 AT %M1017.1 : Bool;
   阀36进指令手动 AT %M1017.4 : Bool;
   阀36回指令手动 AT %M1017.5 : Bool;
   阀37进指令手动 AT %M1018.0 : Bool;
   阀37回指令手动 AT %M1018.1 : Bool;
   阀38进指令手动 AT %M1018.4 : Bool;
   阀38回指令手动 AT %M1018.5 : Bool;
   阀39进指令手动 AT %M1019.0 : Bool;
   阀39回指令手动 AT %M1019.1 : Bool;
   阀40进指令手动 AT %M1019.4 : Bool;
   阀40回指令手动 AT %M1019.5 : Bool;
   阀41进指令手动 AT %M1020.0 : Bool;
   阀41回指令手动 AT %M1020.1 : Bool;
   阀42进指令手动 AT %M1020.4 : Bool;
   阀42回指令手动 AT %M1020.5 : Bool;
   阀43进指令手动 AT %M1021.0 : Bool;
   阀43回指令手动 AT %M1021.1 : Bool;
   阀44进指令手动 AT %M1021.4 : Bool;
   阀44回指令手动 AT %M1021.5 : Bool;
   阀45进指令手动 AT %M1022.0 : Bool;
   阀45回指令手动 AT %M1022.1 : Bool;
   阀46进指令手动 AT %M1022.4 : Bool;
   阀46回指令手动 AT %M1022.5 : Bool;
   阀47进指令手动 AT %M1023.0 : Bool;
   阀47回指令手动 AT %M1023.1 : Bool;
   阀48进指令手动 AT %M1023.4 : Bool;
   阀48回指令手动 AT %M1023.5 : Bool;
   EN_阻挡下到位 AT %M3000.0 : Bool;
   EN_阻挡上到位 AT %M3000.1 : Bool;
   EN_提升机下到位 AT %M3000.4 : Bool;
   EN_提升机上到位 AT %M3000.5 : Bool;
   EX_阻挡下到位 AT %M3001.0 : Bool;
   EX_阻挡上到位 AT %M3001.1 : Bool;
   EX_提升机下到位 AT %M3001.4 : Bool;
   EX_提升机上到位 AT %M3001.5 : Bool;
   ST01上阻挡下到位 AT %M3002.0 : Bool;
   ST01上阻挡上到位 AT %M3002.1 : Bool;
   ST01下阻挡下到位 AT %M3002.4 : Bool;
   ST01下阻挡上到位 AT %M3002.5 : Bool;
   ST02上阻挡下到位 AT %M3003.0 : Bool;
   ST02上阻挡上到位 AT %M3003.1 : Bool;
   ST02下阻挡下到位 AT %M3003.4 : Bool;
   ST02下阻挡上到位 AT %M3003.5 : Bool;
   ST03上阻挡下到位 AT %M3004.0 : Bool;
   ST03上阻挡上到位 AT %M3004.1 : Bool;
   ST03下阻挡下到位 AT %M3004.4 : Bool;
   ST03下阻挡上到位 AT %M3004.5 : Bool;
   ST04上阻挡下到位 AT %M3005.0 : Bool;
   ST04上阻挡上到位 AT %M3005.1 : Bool;
   ST05上阻挡下到位 AT %M3005.4 : Bool;
   ST05上阻挡上到位 AT %M3005.5 : Bool;
   ST06上阻挡下到位 AT %M3006.0 : Bool;
   ST06上阻挡上到位 AT %M3006.1 : Bool;
   ST07上阻挡下到位 AT %M3006.4 : Bool;
   ST07上阻挡上到位 AT %M3006.5 : Bool;
   ST08上阻挡下到位 AT %M3007.0 : Bool;
   ST08上阻挡上到位 AT %M3007.1 : Bool;
   ST09上阻挡下到位 AT %M3007.4 : Bool;
   ST09上阻挡上到位 AT %M3007.5 : Bool;
   ST10上阻挡下到位 AT %M3008.0 : Bool;
   ST10上阻挡上到位 AT %M3008.1 : Bool;
   ST11上阻挡下到位 AT %M3008.4 : Bool;
   ST11上阻挡上到位 AT %M3008.5 : Bool;
   ST12上阻挡下到位 AT %M3009.0 : Bool;
   ST12上阻挡上到位 AT %M3009.1 : Bool;
   阀20进到位 AT %M3009.4 : Bool;
   阀20回到位 AT %M3009.5 : Bool;
   阀21进到位 AT %M3010.0 : Bool;
   阀21回到位 AT %M3010.1 : Bool;
   阀22进到位 AT %M3010.4 : Bool;
   阀22回到位 AT %M3010.5 : Bool;
   阀23进到位 AT %M3011.0 : Bool;
   阀23回到位 AT %M3011.1 : Bool;
   阀24进到位 AT %M3011.4 : Bool;
   阀24回到位 AT %M3011.5 : Bool;
   阀25进到位 AT %M3012.0 : Bool;
   阀25回到位 AT %M3012.1 : Bool;
   阀26进到位 AT %M3012.4 : Bool;
   阀26回到位 AT %M3012.5 : Bool;
   阀27进到位 AT %M3013.0 : Bool;
   阀27回到位 AT %M3013.1 : Bool;
   阀28进到位 AT %M3013.4 : Bool;
   阀28回到位 AT %M3013.5 : Bool;
   阀29进到位 AT %M3014.0 : Bool;
   阀29回到位 AT %M3014.1 : Bool;
   阀30进到位 AT %M3014.4 : Bool;
   阀30回到位 AT %M3014.5 : Bool;
   阀31进到位 AT %M3015.0 : Bool;
   阀31回到位 AT %M3015.1 : Bool;
   阀32进到位 AT %M3015.4 : Bool;
   阀32回到位 AT %M3015.5 : Bool;
   阀33进到位 AT %M3016.0 : Bool;
   阀33回到位 AT %M3016.1 : Bool;
   阀34进到位 AT %M3016.4 : Bool;
   阀34回到位 AT %M3016.5 : Bool;
   阀35进到位 AT %M3017.0 : Bool;
   阀35回到位 AT %M3017.1 : Bool;
   阀36进到位 AT %M3017.4 : Bool;
   阀36回到位 AT %M3017.5 : Bool;
   阀37进到位 AT %M3018.0 : Bool;
   阀37回到位 AT %M3018.1 : Bool;
   阀38进到位 AT %M3018.4 : Bool;
   阀38回到位 AT %M3018.5 : Bool;
   阀39进到位 AT %M3019.0 : Bool;
   阀39回到位 AT %M3019.1 : Bool;
   阀40进到位 AT %M3019.4 : Bool;
   阀40回到位 AT %M3019.5 : Bool;
   阀41进到位 AT %M3020.0 : Bool;
   阀41回到位 AT %M3020.1 : Bool;
   阀42进到位 AT %M3020.4 : Bool;
   阀42回到位 AT %M3020.5 : Bool;
   阀43进到位 AT %M3021.0 : Bool;
   阀43回到位 AT %M3021.1 : Bool;
   阀44进到位 AT %M3021.4 : Bool;
   阀44回到位 AT %M3021.5 : Bool;
   阀45进到位 AT %M3022.0 : Bool;
   阀45回到位 AT %M3022.1 : Bool;
   阀46进到位 AT %M3022.4 : Bool;
   阀46回到位 AT %M3022.5 : Bool;
   阀47进到位 AT %M3023.0 : Bool;
   阀47回到位 AT %M3023.1 : Bool;
   阀48进到位 AT %M3023.4 : Bool;
   阀48回到位 AT %M3023.5 : Bool;
   滚筒1正转指令自动 AT %M2100.0 : Bool;
   滚筒1反转指令自动 AT %M2100.1 : Bool;
   滚筒2正转指令自动 AT %M2100.4 : Bool;
   滚筒2反转指令自动 AT %M2100.5 : Bool;
   滚筒3正转指令自动 AT %M2101.0 : Bool;
   滚筒3反转指令自动 AT %M2101.1 : Bool;
   滚筒4正转指令自动 AT %M2101.4 : Bool;
   滚筒4反转指令自动 AT %M2101.5 : Bool;
   滚筒5正转指令自动 AT %M2102.0 : Bool;
   滚筒5反转指令自动 AT %M2102.1 : Bool;
   滚筒6正转指令自动 AT %M2102.4 : Bool;
   滚筒6反转指令自动 AT %M2102.5 : Bool;
   滚筒7正转指令自动 AT %M2103.0 : Bool;
   滚筒7反转指令自动 AT %M2103.1 : Bool;
   滚筒8正转指令自动 AT %M2103.4 : Bool;
   滚筒8反转指令自动 AT %M2103.5 : Bool;
   滚筒9正转指令自动 AT %M2104.0 : Bool;
   滚筒9反转指令自动 AT %M2104.1 : Bool;
   滚筒10正转指令自动 AT %M2104.4 : Bool;
   滚筒10反转指令自动 AT %M2104.5 : Bool;
   滚筒11正转指令自动 AT %M2105.0 : Bool;
   滚筒11反转指令自动 AT %M2105.1 : Bool;
   滚筒12正转指令自动 AT %M2105.4 : Bool;
   滚筒12反转指令自动 AT %M2105.5 : Bool;
   滚筒13正转指令自动 AT %M2106.0 : Bool;
   滚筒13反转指令自动 AT %M2106.1 : Bool;
   滚筒14正转指令自动 AT %M2106.4 : Bool;
   滚筒14反转指令自动 AT %M2106.5 : Bool;
   滚筒15正转指令自动 AT %M2107.0 : Bool;
   滚筒15反转指令自动 AT %M2107.1 : Bool;
   滚筒16正转指令自动 AT %M2107.4 : Bool;
   滚筒16反转指令自动 AT %M2107.5 : Bool;
   滚筒17正转指令自动 AT %M2108.0 : Bool;
   滚筒17反转指令自动 AT %M2108.1 : Bool;
   滚筒18正转指令自动 AT %M2108.4 : Bool;
   滚筒18反转指令自动 AT %M2108.5 : Bool;
   滚筒19正转指令自动 AT %M2109.0 : Bool;
   滚筒19反转指令自动 AT %M2109.1 : Bool;
   滚筒20正转指令自动 AT %M2109.4 : Bool;
   滚筒20反转指令自动 AT %M2109.5 : Bool;
   滚筒21正转指令自动 AT %M2110.0 : Bool;
   滚筒21反转指令自动 AT %M2110.1 : Bool;
   滚筒22正转指令自动 AT %M2110.4 : Bool;
   滚筒22反转指令自动 AT %M2110.5 : Bool;
   滚筒23正转指令自动 AT %M2111.0 : Bool;
   滚筒23反转指令自动 AT %M2111.1 : Bool;
   滚筒24正转指令自动 AT %M2111.4 : Bool;
   滚筒24反转指令自动 AT %M2111.5 : Bool;
   滚筒25正转指令自动 AT %M2112.0 : Bool;
   滚筒25反转指令自动 AT %M2112.1 : Bool;
   滚筒26正转指令自动 AT %M2112.4 : Bool;
   滚筒26反转指令自动 AT %M2112.5 : Bool;
   滚筒27正转指令自动 AT %M2113.0 : Bool;
   滚筒27反转指令自动 AT %M2113.1 : Bool;
   滚筒28正转指令自动 AT %M2113.4 : Bool;
   滚筒28反转指令自动 AT %M2113.5 : Bool;
   滚筒29正转指令自动 AT %M2114.0 : Bool;
   滚筒29反转指令自动 AT %M2114.1 : Bool;
   滚筒30正转指令自动 AT %M2114.4 : Bool;
   滚筒30反转指令自动 AT %M2114.5 : Bool;
   滚筒31正转指令自动 AT %M2115.0 : Bool;
   滚筒31反转指令自动 AT %M2115.1 : Bool;
   滚筒32正转指令自动 AT %M2115.4 : Bool;
   滚筒32反转指令自动 AT %M2115.5 : Bool;
   滚筒33正转指令自动 AT %M2116.0 : Bool;
   滚筒33反转指令自动 AT %M2116.1 : Bool;
   滚筒34正转指令自动 AT %M2116.4 : Bool;
   滚筒34反转指令自动 AT %M2116.5 : Bool;
   滚筒35正转指令自动 AT %M2117.0 : Bool;
   滚筒35反转指令自动 AT %M2117.1 : Bool;
   滚筒36正转指令自动 AT %M2117.4 : Bool;
   滚筒36反转指令自动 AT %M2117.5 : Bool;
   滚筒37正转指令自动 AT %M2118.0 : Bool;
   滚筒37反转指令自动 AT %M2118.1 : Bool;
   滚筒38正转指令自动 AT %M2118.4 : Bool;
   滚筒38反转指令自动 AT %M2118.5 : Bool;
   滚筒39正转指令自动 AT %M2119.0 : Bool;
   滚筒39反转指令自动 AT %M2119.1 : Bool;
   滚筒40正转指令自动 AT %M2119.4 : Bool;
   滚筒40反转指令自动 AT %M2119.5 : Bool;
   滚筒41正转指令自动 AT %M2120.0 : Bool;
   滚筒41反转指令自动 AT %M2120.1 : Bool;
   滚筒42正转指令自动 AT %M2120.4 : Bool;
   滚筒42反转指令自动 AT %M2120.5 : Bool;
   滚筒43正转指令自动 AT %M2121.0 : Bool;
   滚筒43反转指令自动 AT %M2121.1 : Bool;
   滚筒44正转指令自动 AT %M2121.4 : Bool;
   滚筒44反转指令自动 AT %M2121.5 : Bool;
   滚筒45正转指令自动 AT %M2122.0 : Bool;
   滚筒45反转指令自动 AT %M2122.1 : Bool;
   滚筒46正转指令自动 AT %M2122.4 : Bool;
   滚筒46反转指令自动 AT %M2122.5 : Bool;
   滚筒47正转指令自动 AT %M2123.0 : Bool;
   滚筒47反转指令自动 AT %M2123.1 : Bool;
   滚筒48正转指令自动 AT %M2123.4 : Bool;
   滚筒48反转指令自动 AT %M2123.5 : Bool;
   滚筒1正转指令手动 AT %M1100.0 : Bool;
   滚筒1反转指令手动 AT %M1100.1 : Bool;
   滚筒2正转指令手动 AT %M1100.4 : Bool;
   滚筒2反转指令手动 AT %M1100.5 : Bool;
   滚筒3正转指令手动 AT %M1101.0 : Bool;
   滚筒3反转指令手动 AT %M1101.1 : Bool;
   滚筒4正转指令手动 AT %M1101.4 : Bool;
   滚筒4反转指令手动 AT %M1101.5 : Bool;
   滚筒5正转指令手动 AT %M1102.0 : Bool;
   滚筒5反转指令手动 AT %M1102.1 : Bool;
   滚筒6正转指令手动 AT %M1102.4 : Bool;
   滚筒6反转指令手动 AT %M1102.5 : Bool;
   滚筒7正转指令手动 AT %M1103.0 : Bool;
   滚筒7反转指令手动 AT %M1103.1 : Bool;
   滚筒8正转指令手动 AT %M1103.4 : Bool;
   滚筒8反转指令手动 AT %M1103.5 : Bool;
   滚筒9正转指令手动 AT %M1104.0 : Bool;
   滚筒9反转指令手动 AT %M1104.1 : Bool;
   滚筒10正转指令手动 AT %M1104.4 : Bool;
   滚筒10反转指令手动 AT %M1104.5 : Bool;
   滚筒11正转指令手动 AT %M1105.0 : Bool;
   滚筒11反转指令手动 AT %M1105.1 : Bool;
   滚筒12正转指令手动 AT %M1105.4 : Bool;
   滚筒12反转指令手动 AT %M1105.5 : Bool;
   滚筒13正转指令手动 AT %M1106.0 : Bool;
   滚筒13反转指令手动 AT %M1106.1 : Bool;
   滚筒14正转指令手动 AT %M1106.4 : Bool;
   滚筒14反转指令手动 AT %M1106.5 : Bool;
   滚筒15正转指令手动 AT %M1107.0 : Bool;
   滚筒15反转指令手动 AT %M1107.1 : Bool;
   滚筒16正转指令手动 AT %M1107.4 : Bool;
   滚筒16反转指令手动 AT %M1107.5 : Bool;
   滚筒17正转指令手动 AT %M1108.0 : Bool;
   滚筒17反转指令手动 AT %M1108.1 : Bool;
   滚筒18正转指令手动 AT %M1108.4 : Bool;
   滚筒18反转指令手动 AT %M1108.5 : Bool;
   滚筒19正转指令手动 AT %M1109.0 : Bool;
   滚筒19反转指令手动 AT %M1109.1 : Bool;
   滚筒20正转指令手动 AT %M1109.4 : Bool;
   滚筒20反转指令手动 AT %M1109.5 : Bool;
   滚筒21正转指令手动 AT %M1110.0 : Bool;
   滚筒21反转指令手动 AT %M1110.1 : Bool;
   滚筒22正转指令手动 AT %M1110.4 : Bool;
   滚筒22反转指令手动 AT %M1110.5 : Bool;
   滚筒23正转指令手动 AT %M1111.0 : Bool;
   滚筒23反转指令手动 AT %M1111.1 : Bool;
   滚筒24正转指令手动 AT %M1111.4 : Bool;
   滚筒24反转指令手动 AT %M1111.5 : Bool;
   滚筒25正转指令手动 AT %M1112.0 : Bool;
   滚筒25反转指令手动 AT %M1112.1 : Bool;
   滚筒26正转指令手动 AT %M1112.4 : Bool;
   滚筒26反转指令手动 AT %M1112.5 : Bool;
   滚筒27正转指令手动 AT %M1113.0 : Bool;
   滚筒27反转指令手动 AT %M1113.1 : Bool;
   滚筒28正转指令手动 AT %M1113.4 : Bool;
   滚筒28反转指令手动 AT %M1113.5 : Bool;
   滚筒29正转指令手动 AT %M1114.0 : Bool;
   滚筒29反转指令手动 AT %M1114.1 : Bool;
   滚筒30正转指令手动 AT %M1114.4 : Bool;
   滚筒30反转指令手动 AT %M1114.5 : Bool;
   滚筒31正转指令手动 AT %M1115.0 : Bool;
   滚筒31反转指令手动 AT %M1115.1 : Bool;
   滚筒32正转指令手动 AT %M1115.4 : Bool;
   滚筒32反转指令手动 AT %M1115.5 : Bool;
   滚筒33正转指令手动 AT %M1116.0 : Bool;
   滚筒33反转指令手动 AT %M1116.1 : Bool;
   滚筒34正转指令手动 AT %M1116.4 : Bool;
   滚筒34反转指令手动 AT %M1116.5 : Bool;
   滚筒35正转指令手动 AT %M1117.0 : Bool;
   滚筒35反转指令手动 AT %M1117.1 : Bool;
   滚筒36正转指令手动 AT %M1117.4 : Bool;
   滚筒36反转指令手动 AT %M1117.5 : Bool;
   滚筒37正转指令手动 AT %M1118.0 : Bool;
   滚筒37反转指令手动 AT %M1118.1 : Bool;
   滚筒38正转指令手动 AT %M1118.4 : Bool;
   滚筒38反转指令手动 AT %M1118.5 : Bool;
   滚筒39正转指令手动 AT %M1119.0 : Bool;
   滚筒39反转指令手动 AT %M1119.1 : Bool;
   滚筒40正转指令手动 AT %M1119.4 : Bool;
   滚筒40反转指令手动 AT %M1119.5 : Bool;
   滚筒41正转指令手动 AT %M1120.0 : Bool;
   滚筒41反转指令手动 AT %M1120.1 : Bool;
   滚筒42正转指令手动 AT %M1120.4 : Bool;
   滚筒42反转指令手动 AT %M1120.5 : Bool;
   滚筒43正转指令手动 AT %M1121.0 : Bool;
   滚筒43反转指令手动 AT %M1121.1 : Bool;
   滚筒44正转指令手动 AT %M1121.4 : Bool;
   滚筒44反转指令手动 AT %M1121.5 : Bool;
   滚筒45正转指令手动 AT %M1122.0 : Bool;
   滚筒45反转指令手动 AT %M1122.1 : Bool;
   滚筒46正转指令手动 AT %M1122.4 : Bool;
   滚筒46反转指令手动 AT %M1122.5 : Bool;
   滚筒47正转指令手动 AT %M1123.0 : Bool;
   滚筒47反转指令手动 AT %M1123.1 : Bool;
   滚筒48正转指令手动 AT %M1123.4 : Bool;
   滚筒48反转指令手动 AT %M1123.5 : Bool;
   "滚筒1正转到位(不用" AT %M3100.0 : Bool;
   "滚筒1反转到位(不用" AT %M3100.1 : Bool;
   "滚筒2正转到位(不用" AT %M3100.4 : Bool;
   "滚筒2反转到位(不用" AT %M3100.5 : Bool;
   "滚筒3正转到位(不用" AT %M3101.0 : Bool;
   "滚筒3反转到位(不用" AT %M3101.1 : Bool;
   "滚筒4正转到位(不用" AT %M3101.4 : Bool;
   "滚筒4反转到位(不用" AT %M3101.5 : Bool;
   "滚筒5正转到位(不用" AT %M3102.0 : Bool;
   "滚筒5反转到位(不用" AT %M3102.1 : Bool;
   "滚筒6正转到位(不用" AT %M3102.4 : Bool;
   "滚筒6反转到位(不用" AT %M3102.5 : Bool;
   "滚筒7正转到位(不用" AT %M3103.0 : Bool;
   "滚筒7反转到位(不用" AT %M3103.1 : Bool;
   "滚筒8正转到位(不用" AT %M3103.4 : Bool;
   "滚筒8反转到位(不用" AT %M3103.5 : Bool;
   "滚筒9正转到位(不用" AT %M3104.0 : Bool;
   "滚筒9反转到位(不用" AT %M3104.1 : Bool;
   "滚筒10正转到位(不用" AT %M3104.4 : Bool;
   "滚筒10反转到位(不用" AT %M3104.5 : Bool;
   "滚筒11正转到位(不用" AT %M3105.0 : Bool;
   "滚筒11反转到位(不用" AT %M3105.1 : Bool;
   "滚筒12正转到位(不用" AT %M3105.4 : Bool;
   "滚筒12反转到位(不用" AT %M3105.5 : Bool;
   "滚筒13正转到位(不用" AT %M3106.0 : Bool;
   "滚筒13反转到位(不用" AT %M3106.1 : Bool;
   "滚筒14正转到位(不用" AT %M3106.4 : Bool;
   "滚筒14反转到位(不用" AT %M3106.5 : Bool;
   "滚筒15正转到位(不用" AT %M3107.0 : Bool;
   "滚筒15反转到位(不用" AT %M3107.1 : Bool;
   "滚筒16正转到位(不用" AT %M3107.4 : Bool;
   "滚筒16反转到位(不用" AT %M3107.5 : Bool;
   "滚筒17正转到位(不用" AT %M3108.0 : Bool;
   "滚筒17反转到位(不用" AT %M3108.1 : Bool;
   "滚筒18正转到位(不用" AT %M3108.4 : Bool;
   "滚筒18反转到位(不用" AT %M3108.5 : Bool;
   "滚筒19正转到位(不用" AT %M3109.0 : Bool;
   "滚筒19反转到位(不用" AT %M3109.1 : Bool;
   "滚筒20正转到位(不用" AT %M3109.4 : Bool;
   "滚筒20反转到位(不用" AT %M3109.5 : Bool;
   "滚筒21正转到位(不用" AT %M3110.0 : Bool;
   "滚筒21反转到位(不用" AT %M3110.1 : Bool;
   "滚筒22正转到位(不用" AT %M3110.4 : Bool;
   "滚筒22反转到位(不用" AT %M3110.5 : Bool;
   "滚筒23正转到位(不用" AT %M3111.0 : Bool;
   "滚筒23反转到位(不用" AT %M3111.1 : Bool;
   "滚筒24正转到位(不用" AT %M3111.4 : Bool;
   "滚筒24反转到位(不用" AT %M3111.5 : Bool;
   "滚筒25正转到位(不用" AT %M3112.0 : Bool;
   "滚筒25反转到位(不用" AT %M3112.1 : Bool;
   "滚筒26正转到位(不用" AT %M3112.4 : Bool;
   "滚筒26反转到位(不用" AT %M3112.5 : Bool;
   "滚筒27正转到位(不用" AT %M3113.0 : Bool;
   "滚筒27反转到位(不用" AT %M3113.1 : Bool;
   "滚筒28正转到位(不用" AT %M3113.4 : Bool;
   "滚筒28反转到位(不用" AT %M3113.5 : Bool;
   "滚筒29正转到位(不用" AT %M3114.0 : Bool;
   "滚筒29反转到位(不用" AT %M3114.1 : Bool;
   "滚筒30正转到位(不用" AT %M3114.4 : Bool;
   "滚筒30反转到位(不用" AT %M3114.5 : Bool;
   "滚筒31正转到位(不用" AT %M3115.0 : Bool;
   "滚筒31反转到位(不用" AT %M3115.1 : Bool;
   "滚筒32正转到位(不用" AT %M3115.4 : Bool;
   "滚筒32反转到位(不用" AT %M3115.5 : Bool;
   "滚筒33正转到位(不用" AT %M3116.0 : Bool;
   "滚筒33反转到位(不用" AT %M3116.1 : Bool;
   "滚筒34正转到位(不用" AT %M3116.4 : Bool;
   "滚筒34反转到位(不用" AT %M3116.5 : Bool;
   "滚筒35正转到位(不用" AT %M3117.0 : Bool;
   "滚筒35反转到位(不用" AT %M3117.1 : Bool;
   "滚筒36正转到位(不用" AT %M3117.4 : Bool;
   "滚筒36反转到位(不用" AT %M3117.5 : Bool;
   "滚筒37正转到位(不用" AT %M3118.0 : Bool;
   "滚筒37反转到位(不用" AT %M3118.1 : Bool;
   "滚筒38正转到位(不用" AT %M3118.4 : Bool;
   "滚筒38反转到位(不用" AT %M3118.5 : Bool;
   "滚筒39正转到位(不用" AT %M3119.0 : Bool;
   "滚筒39反转到位(不用" AT %M3119.1 : Bool;
   "滚筒40正转到位(不用" AT %M3119.4 : Bool;
   "滚筒40反转到位(不用" AT %M3119.5 : Bool;
   "滚筒41正转到位(不用" AT %M3120.0 : Bool;
   "滚筒41反转到位(不用" AT %M3120.1 : Bool;
   "滚筒42正转到位(不用" AT %M3120.4 : Bool;
   "滚筒42反转到位(不用" AT %M3120.5 : Bool;
   "滚筒43正转到位(不用" AT %M3121.0 : Bool;
   "滚筒43反转到位(不用" AT %M3121.1 : Bool;
   "滚筒44正转到位(不用" AT %M3121.4 : Bool;
   "滚筒44反转到位(不用" AT %M3121.5 : Bool;
   "滚筒45正转到位(不用" AT %M3122.0 : Bool;
   "滚筒45反转到位(不用" AT %M3122.1 : Bool;
   "滚筒46正转到位(不用" AT %M3122.4 : Bool;
   "滚筒46反转到位(不用" AT %M3122.5 : Bool;
   "滚筒47正转到位(不用" AT %M3123.0 : Bool;
   "滚筒47反转到位(不用" AT %M3123.1 : Bool;
   "滚筒48正转到位(不用" AT %M3123.4 : Bool;
   "滚筒48反转到位(不用" AT %M3123.5 : Bool;
   变频器1正转指令自动 AT %M2200.0 : Bool;
   变频器1反转指令自动 AT %M2200.1 : Bool;
   变频器2正转指令自动 AT %M2200.4 : Bool;
   变频器2反转指令自动 AT %M2200.5 : Bool;
   变频器3正转指令自动 AT %M2201.0 : Bool;
   变频器3反转指令自动 AT %M2201.1 : Bool;
   变频器4正转指令自动 AT %M2201.4 : Bool;
   变频器4反转指令自动 AT %M2201.5 : Bool;
   变频器5正转指令自动 AT %M2202.0 : Bool;
   变频器5反转指令自动 AT %M2202.1 : Bool;
   变频器6正转指令自动 AT %M2202.4 : Bool;
   变频器6反转指令自动 AT %M2202.5 : Bool;
   变频器7正转指令自动 AT %M2203.0 : Bool;
   变频器7反转指令自动 AT %M2203.1 : Bool;
   变频器8正转指令自动 AT %M2203.4 : Bool;
   变频器8反转指令自动 AT %M2203.5 : Bool;
   变频器9正转指令自动 AT %M2204.0 : Bool;
   变频器9反转指令自动 AT %M2204.1 : Bool;
   变频器10正转指令自动 AT %M2204.4 : Bool;
   变频器10反转指令自动 AT %M2204.5 : Bool;
   变频器11正转指令自动 AT %M2205.0 : Bool;
   变频器11反转指令自动 AT %M2205.1 : Bool;
   变频器12正转指令自动 AT %M2205.4 : Bool;
   变频器12反转指令自动 AT %M2205.5 : Bool;
   变频器13正转指令自动 AT %M2206.0 : Bool;
   变频器13反转指令自动 AT %M2206.1 : Bool;
   变频器14正转指令自动 AT %M2206.4 : Bool;
   变频器14反转指令自动 AT %M2206.5 : Bool;
   变频器15正转指令自动 AT %M2207.0 : Bool;
   变频器15反转指令自动 AT %M2207.1 : Bool;
   变频器16正转指令自动 AT %M2207.4 : Bool;
   变频器16反转指令自动 AT %M2207.5 : Bool;
   变频器1正转指令手动 AT %M1200.0 : Bool;
   变频器1反转指令手动 AT %M1200.1 : Bool;
   变频器2正转指令手动 AT %M1200.4 : Bool;
   变频器2反转指令手动 AT %M1200.5 : Bool;
   变频器3正转指令手动 AT %M1201.0 : Bool;
   变频器3反转指令手动 AT %M1201.1 : Bool;
   变频器4正转指令手动 AT %M1201.4 : Bool;
   变频器4反转指令手动 AT %M1201.5 : Bool;
   变频器5正转指令手动 AT %M1202.0 : Bool;
   变频器5反转指令手动 AT %M1202.1 : Bool;
   变频器6正转指令手动 AT %M1202.4 : Bool;
   变频器6反转指令手动 AT %M1202.5 : Bool;
   变频器7正转指令手动 AT %M1203.0 : Bool;
   变频器7反转指令手动 AT %M1203.1 : Bool;
   变频器8正转指令手动 AT %M1203.4 : Bool;
   变频器8反转指令手动 AT %M1203.5 : Bool;
   变频器9正转指令手动 AT %M1204.0 : Bool;
   变频器9反转指令手动 AT %M1204.1 : Bool;
   变频器10正转指令手动 AT %M1204.4 : Bool;
   变频器10反转指令手动 AT %M1204.5 : Bool;
   变频器11正转指令手动 AT %M1205.0 : Bool;
   变频器11反转指令手动 AT %M1205.1 : Bool;
   变频器12正转指令手动 AT %M1205.4 : Bool;
   变频器12反转指令手动 AT %M1205.5 : Bool;
   变频器13正转指令手动 AT %M1206.0 : Bool;
   变频器13反转指令手动 AT %M1206.1 : Bool;
   变频器14正转指令手动 AT %M1206.4 : Bool;
   变频器14反转指令手动 AT %M1206.5 : Bool;
   变频器15正转指令手动 AT %M1207.0 : Bool;
   变频器15反转指令手动 AT %M1207.1 : Bool;
   变频器16正转指令手动 AT %M1207.4 : Bool;
   变频器16反转指令手动 AT %M1207.5 : Bool;
   "变频器1正转到位(不用" AT %M3200.0 : Bool;
   "变频器1反转到位(不用" AT %M3200.1 : Bool;
   "变频器2正转到位(不用" AT %M3200.4 : Bool;
   "变频器2反转到位(不用" AT %M3200.5 : Bool;
   "变频器3正转到位(不用" AT %M3201.0 : Bool;
   "变频器3反转到位(不用" AT %M3201.1 : Bool;
   "变频器4正转到位(不用" AT %M3201.4 : Bool;
   "变频器4反转到位(不用" AT %M3201.5 : Bool;
   "变频器5正转到位(不用" AT %M3202.0 : Bool;
   "变频器5反转到位(不用" AT %M3202.1 : Bool;
   "变频器6正转到位(不用" AT %M3202.4 : Bool;
   "变频器6反转到位(不用" AT %M3202.5 : Bool;
   "变频器7正转到位(不用" AT %M3203.0 : Bool;
   "变频器7反转到位(不用" AT %M3203.1 : Bool;
   "变频器8正转到位(不用" AT %M3203.4 : Bool;
   "变频器8反转到位(不用" AT %M3203.5 : Bool;
   "变频器9正转到位(不用" AT %M3204.0 : Bool;
   "变频器9反转到位(不用" AT %M3204.1 : Bool;
   "变频器10正转到位(不用" AT %M3204.4 : Bool;
   "变频器10反转到位(不用" AT %M3204.5 : Bool;
   "变频器11正转到位(不用" AT %M3205.0 : Bool;
   "变频器11反转到位(不用" AT %M3205.1 : Bool;
   "变频器12正转到位(不用" AT %M3205.4 : Bool;
   "变频器12反转到位(不用" AT %M3205.5 : Bool;
   "变频器13正转到位(不用" AT %M3206.0 : Bool;
   "变频器13反转到位(不用" AT %M3206.1 : Bool;
   "变频器14正转到位(不用" AT %M3206.4 : Bool;
   "变频器14反转到位(不用" AT %M3206.5 : Bool;
   "变频器15正转到位(不用" AT %M3207.0 : Bool;
   "变频器15反转到位(不用" AT %M3207.1 : Bool;
   "变频器16正转到位(不用" AT %M3207.4 : Bool;
   "变频器16反转到位(不用" AT %M3207.5 : Bool;
END_VAR

VAR_GLOBAL   // PLC tag table "106轴控制变量表"
   轴1定位1自动 AT %M2400.0 : Bool;
   轴1定位2自动 AT %M2400.1 : Bool;
   轴1定位3自动 AT %M2400.2 : Bool;
   轴1定位4自动 AT %M2400.3 : Bool;
   轴1xx1 AT %M2400.4 : Bool;
   轴1xx2 AT %M2400.5 : Bool;
   轴1xx3 AT %M2400.6 : Bool;
   轴1xx4 AT %M2400.7 : Bool;
   轴2定位1自动 AT %M2402.0 : Bool;
   轴2定位2自动 AT %M2402.1 : Bool;
   轴2定位3自动 AT %M2402.2 : Bool;
   轴2定位4自动 AT %M2402.3 : Bool;
   轴2xx1 AT %M2402.4 : Bool;
   轴2xx2 AT %M2402.5 : Bool;
   轴2xx3 AT %M2402.6 : Bool;
   轴2xx4 AT %M2402.7 : Bool;
   轴3定位1自动 AT %M2404.0 : Bool;
   轴3定位2自动 AT %M2404.1 : Bool;
   轴3定位3自动 AT %M2404.2 : Bool;
   轴3定位4自动 AT %M2404.3 : Bool;
   轴3xx1 AT %M2404.4 : Bool;
   轴3xx2 AT %M2404.5 : Bool;
   轴3xx3 AT %M2404.6 : Bool;
   轴3xx4 AT %M2404.7 : Bool;
   轴4定位1自动 AT %M2406.0 : Bool;
   轴4定位2自动 AT %M2406.1 : Bool;
   轴4定位3自动 AT %M2406.2 : Bool;
   轴4定位4自动 AT %M2406.3 : Bool;
   轴4xx1 AT %M2406.4 : Bool;
   轴4xx2 AT %M2406.5 : Bool;
   轴4xx3 AT %M2406.6 : Bool;
   轴4xx4 AT %M2406.7 : Bool;
   轴5定位1自动 AT %M2408.0 : Bool;
   轴5定位2自动 AT %M2408.1 : Bool;
   轴5定位3自动 AT %M2408.2 : Bool;
   轴5定位4自动 AT %M2408.3 : Bool;
   轴5xx1 AT %M2408.4 : Bool;
   轴5xx2 AT %M2408.5 : Bool;
   轴5xx3 AT %M2408.6 : Bool;
   轴5xx4 AT %M2408.7 : Bool;
   轴6定位1自动 AT %M2410.0 : Bool;
   轴6定位2自动 AT %M2410.1 : Bool;
   轴6定位3自动 AT %M2410.2 : Bool;
   轴6定位4自动 AT %M2410.3 : Bool;
   轴6xx1 AT %M2410.4 : Bool;
   轴6xx2 AT %M2410.5 : Bool;
   轴6xx3 AT %M2410.6 : Bool;
   轴6xx4 AT %M2410.7 : Bool;
   轴7定位1自动 AT %M2412.0 : Bool;
   轴7定位2自动 AT %M2412.1 : Bool;
   轴7定位3自动 AT %M2412.2 : Bool;
   轴7定位4自动 AT %M2412.3 : Bool;
   轴7xx1 AT %M2412.4 : Bool;
   轴7xx2 AT %M2412.5 : Bool;
   轴7xx3 AT %M2412.6 : Bool;
   轴7xx4 AT %M2412.7 : Bool;
   轴8定位1自动 AT %M2414.0 : Bool;
   轴8定位2自动 AT %M2414.1 : Bool;
   轴8定位3自动 AT %M2414.2 : Bool;
   轴8定位4自动 AT %M2414.3 : Bool;
   轴8xx1 AT %M2414.4 : Bool;
   轴8xx2 AT %M2414.5 : Bool;
   轴8xx3 AT %M2414.6 : Bool;
   轴8xx4 AT %M2414.7 : Bool;
   轴9定位1自动 AT %M2416.0 : Bool;
   轴9定位2自动 AT %M2416.1 : Bool;
   轴9定位3自动 AT %M2416.2 : Bool;
   轴9定位4自动 AT %M2416.3 : Bool;
   轴9xx1 AT %M2416.4 : Bool;
   轴9xx2 AT %M2416.5 : Bool;
   轴9xx3 AT %M2416.6 : Bool;
   轴9xx4 AT %M2416.7 : Bool;
   轴10定位1自动 AT %M2418.0 : Bool;
   轴10定位2自动 AT %M2418.1 : Bool;
   轴10定位3自动 AT %M2418.2 : Bool;
   轴10定位4自动 AT %M2418.3 : Bool;
   轴10xx1 AT %M2418.4 : Bool;
   轴10xx2 AT %M2418.5 : Bool;
   轴10xx3 AT %M2418.6 : Bool;
   轴10xx4 AT %M2418.7 : Bool;
   轴11定位1自动 AT %M2420.0 : Bool;
   轴11定位2自动 AT %M2420.1 : Bool;
   轴11定位3自动 AT %M2420.2 : Bool;
   轴11定位4自动 AT %M2420.3 : Bool;
   轴11xx1 AT %M2420.4 : Bool;
   轴11xx2 AT %M2420.5 : Bool;
   轴11xx3 AT %M2420.6 : Bool;
   轴11xx4 AT %M2420.7 : Bool;
   轴12定位1自动 AT %M2422.0 : Bool;
   轴12定位2自动 AT %M2422.1 : Bool;
   轴12定位3自动 AT %M2422.2 : Bool;
   轴12定位4自动 AT %M2422.3 : Bool;
   轴12xx1 AT %M2422.4 : Bool;
   轴12xx2 AT %M2422.5 : Bool;
   轴12xx3 AT %M2422.6 : Bool;
   轴12xx4 AT %M2422.7 : Bool;
   轴13定位1自动 AT %M2424.0 : Bool;
   轴13定位2自动 AT %M2424.1 : Bool;
   轴13定位3自动 AT %M2424.2 : Bool;
   轴13定位4自动 AT %M2424.3 : Bool;
   轴13xx1 AT %M2424.4 : Bool;
   轴13xx2 AT %M2424.5 : Bool;
   轴13xx3 AT %M2424.6 : Bool;
   轴13xx4 AT %M2424.7 : Bool;
   轴14定位1自动 AT %M2426.0 : Bool;
   轴14定位2自动 AT %M2426.1 : Bool;
   轴14定位3自动 AT %M2426.2 : Bool;
   轴14定位4自动 AT %M2426.3 : Bool;
   轴14xx1 AT %M2426.4 : Bool;
   轴14xx2 AT %M2426.5 : Bool;
   轴14xx3 AT %M2426.6 : Bool;
   轴14xx4 AT %M2426.7 : Bool;
   轴15定位1自动 AT %M2428.0 : Bool;
   轴15定位2自动 AT %M2428.1 : Bool;
   轴15定位3自动 AT %M2428.2 : Bool;
   轴15定位4自动 AT %M2428.3 : Bool;
   轴15xx1 AT %M2428.4 : Bool;
   轴15xx2 AT %M2428.5 : Bool;
   轴15xx3 AT %M2428.6 : Bool;
   轴15xx4 AT %M2428.7 : Bool;
   轴16定位1自动 AT %M2430.0 : Bool;
   轴16定位2自动 AT %M2430.1 : Bool;
   轴16定位3自动 AT %M2430.2 : Bool;
   轴16定位4自动 AT %M2430.3 : Bool;
   轴16xx1 AT %M2430.4 : Bool;
   轴16xx2 AT %M2430.5 : Bool;
   轴16xx3 AT %M2430.6 : Bool;
   轴16xx4 AT %M2430.7 : Bool;
   XXXXXX1 AT %M2432.0 : Bool;
   轴1定位1手动 AT %M1400.0 : Bool;
   轴1定位2手动 AT %M1400.1 : Bool;
   轴1定位3手动 AT %M1400.2 : Bool;
   轴1定位4手动 AT %M1400.3 : Bool;
   轴1xx1手动 AT %M1400.4 : Bool;
   轴1xx2手动 AT %M1400.5 : Bool;
   轴1xx3手动 AT %M1400.6 : Bool;
   轴1xx4手动 AT %M1400.7 : Bool;
   轴1使能 AT %M1401.0 : Bool;
   轴1回零 AT %M1401.1 : Bool;
   "轴1点动+" AT %M1401.2 : Bool;
   "轴1点动-" AT %M1401.3 : Bool;
   轴1自由定位 AT %M1401.4 : Bool;
   轴1就绪 AT %M1401.5 : Bool;
   轴1原点 AT %M1401.6 : Bool;
   轴1到达 AT %M1401.7 : Bool;
   轴2定位1手动 AT %M1402.0 : Bool;
   轴2定位2手动 AT %M1402.1 : Bool;
   轴2定位3手动 AT %M1402.2 : Bool;
   轴2定位4手动 AT %M1402.3 : Bool;
   轴2xx1手动 AT %M1402.4 : Bool;
   轴2xx2手动 AT %M1402.5 : Bool;
   轴2xx3手动 AT %M1402.6 : Bool;
   轴2xx4手动 AT %M1402.7 : Bool;
   轴2使能 AT %M1403.0 : Bool;
   轴2回零 AT %M1403.1 : Bool;
   "轴2点动+" AT %M1403.2 : Bool;
   "轴2点动-" AT %M1403.3 : Bool;
   轴2自由定位 AT %M1403.4 : Bool;
   轴2就绪 AT %M1403.5 : Bool;
   轴2原点 AT %M1403.6 : Bool;
   轴2到达 AT %M1403.7 : Bool;
   轴3定位1手动 AT %M1404.0 : Bool;
   轴3定位2手动 AT %M1404.1 : Bool;
   轴3定位3手动 AT %M1404.2 : Bool;
   轴3定位4手动 AT %M1404.3 : Bool;
   轴3xx1手动 AT %M1404.4 : Bool;
   轴3xx2手动 AT %M1404.5 : Bool;
   轴3xx3手动 AT %M1404.6 : Bool;
   轴3xx4手动 AT %M1404.7 : Bool;
   轴3使能 AT %M1405.0 : Bool;
   轴3回零 AT %M1405.1 : Bool;
   "轴3点动+" AT %M1405.2 : Bool;
   "轴3点动-" AT %M1405.3 : Bool;
   轴3自由定位 AT %M1405.4 : Bool;
   轴3就绪 AT %M1405.5 : Bool;
   轴3原点 AT %M1405.6 : Bool;
   轴3到达 AT %M1405.7 : Bool;
   轴4定位1手动 AT %M1406.0 : Bool;
   轴4定位2手动 AT %M1406.1 : Bool;
   轴4定位3手动 AT %M1406.2 : Bool;
   轴4自由定位 AT %M1407.4 : Bool;
   轴4xx1手动 AT %M1406.4 : Bool;
   轴4xx2手动 AT %M1406.5 : Bool;
   轴4xx3手动 AT %M1406.6 : Bool;
   轴4xx4手动 AT %M1406.7 : Bool;
   轴4使能 AT %M1407.0 : Bool;
   轴4回零 AT %M1407.1 : Bool;
   "轴4点动+" AT %M1407.2 : Bool;
   "轴4点动-" AT %M1407.3 : Bool;
   轴4就绪 AT %M1407.5 : Bool;
   轴4原点 AT %M1407.6 : Bool;
   轴4到达 AT %M1407.7 : Bool;
   轴5定位1手动 AT %M1408.0 : Bool;
   轴5定位2手动 AT %M1408.1 : Bool;
   轴5定位3手动 AT %M1408.2 : Bool;
   轴5定位4手动 AT %M1408.3 : Bool;
   轴5xx1手动 AT %M1408.4 : Bool;
   轴5xx2手动 AT %M1408.5 : Bool;
   轴5xx3手动 AT %M1408.6 : Bool;
   轴5xx4手动 AT %M1408.7 : Bool;
   轴5使能 AT %M1409.0 : Bool;
   轴5回零 AT %M1409.1 : Bool;
   "轴5点动+" AT %M1409.2 : Bool;
   "轴5点动-" AT %M1409.3 : Bool;
   轴5自由定位 AT %M1409.4 : Bool;
   轴5就绪 AT %M1409.5 : Bool;
   轴5原点 AT %M1409.6 : Bool;
   轴5到达 AT %M1409.7 : Bool;
   轴6定位1手动 AT %M1410.0 : Bool;
   轴6定位2手动 AT %M1410.1 : Bool;
   轴6定位3手动 AT %M1410.2 : Bool;
   轴6定位4手动 AT %M1410.3 : Bool;
   轴6xx1手动 AT %M1410.4 : Bool;
   轴6xx2手动 AT %M1410.5 : Bool;
   轴6xx3手动 AT %M1410.6 : Bool;
   轴6xx4手动 AT %M1410.7 : Bool;
   轴6使能 AT %M1411.0 : Bool;
   轴6回零 AT %M1411.1 : Bool;
   "轴6点动+" AT %M1411.2 : Bool;
   "轴6点动-" AT %M1411.3 : Bool;
   轴6自由定位 AT %M1411.4 : Bool;
   轴6就绪 AT %M1411.5 : Bool;
   轴6原点 AT %M1411.6 : Bool;
   轴6到达 AT %M1411.7 : Bool;
   轴7定位1手动 AT %M1412.0 : Bool;
   轴7定位2手动 AT %M1412.1 : Bool;
   轴7定位3手动 AT %M1412.2 : Bool;
   轴7定位4手动 AT %M1412.3 : Bool;
   轴7xx1手动 AT %M1412.4 : Bool;
   轴7xx2手动 AT %M1412.5 : Bool;
   轴7xx3手动 AT %M1412.6 : Bool;
   轴7xx4手动 AT %M1412.7 : Bool;
   轴7使能 AT %M1413.0 : Bool;
   轴7回零 AT %M1413.1 : Bool;
   "轴7点动+" AT %M1413.2 : Bool;
   "轴7点动-" AT %M1413.3 : Bool;
   轴7自由定位 AT %M1413.4 : Bool;
   轴7就绪 AT %M1413.5 : Bool;
   轴7原点 AT %M1413.6 : Bool;
   轴7到达 AT %M1413.7 : Bool;
   轴8定位1手动 AT %M1414.0 : Bool;
   轴8定位2手动 AT %M1414.1 : Bool;
   轴8定位3手动 AT %M1414.2 : Bool;
   轴8定位4手动 AT %M1414.3 : Bool;
   轴8xx1手动 AT %M1414.4 : Bool;
   轴8xx2手动 AT %M1414.5 : Bool;
   轴8xx3手动 AT %M1414.6 : Bool;
   轴8xx4手动 AT %M1414.7 : Bool;
   轴8使能 AT %M1415.0 : Bool;
   轴8回零 AT %M1415.1 : Bool;
   "轴8点动+" AT %M1415.2 : Bool;
   "轴8点动-" AT %M1415.3 : Bool;
   轴8自由定位 AT %M1415.4 : Bool;
   轴8就绪 AT %M1415.5 : Bool;
   轴8原点 AT %M1415.6 : Bool;
   轴8到达 AT %M1415.7 : Bool;
   轴9定位1手动 AT %M1416.0 : Bool;
   轴9定位2手动 AT %M1416.1 : Bool;
   轴9定位3手动 AT %M1416.2 : Bool;
   轴9定位4手动 AT %M1416.3 : Bool;
   轴9xx1手动 AT %M1416.4 : Bool;
   轴9xx2手动 AT %M1416.5 : Bool;
   轴9xx3手动 AT %M1416.6 : Bool;
   轴9xx4手动 AT %M1416.7 : Bool;
   轴9使能 AT %M1417.0 : Bool;
   轴9回零 AT %M1417.1 : Bool;
   "轴9点动+" AT %M1417.2 : Bool;
   "轴9点动-" AT %M1417.3 : Bool;
   轴9自由定位 AT %M1417.4 : Bool;
   轴9就绪 AT %M1417.5 : Bool;
   轴9原点 AT %M1417.6 : Bool;
   轴9到达 AT %M1417.7 : Bool;
   轴10定位1手动 AT %M1418.0 : Bool;
   轴10定位2手动 AT %M1418.1 : Bool;
   轴10定位3手动 AT %M1418.2 : Bool;
   轴10定位4手动 AT %M1418.3 : Bool;
   轴10xx1手动 AT %M1418.4 : Bool;
   轴10xx2手动 AT %M1418.5 : Bool;
   轴10xx3手动 AT %M1418.6 : Bool;
   轴10xx4手动 AT %M1418.7 : Bool;
   轴10使能 AT %M1419.0 : Bool;
   轴10回零 AT %M1419.1 : Bool;
   "轴10点动+" AT %M1419.2 : Bool;
   "轴10点动-" AT %M1419.3 : Bool;
   轴10自由定位 AT %M1419.4 : Bool;
   轴10就绪 AT %M1419.5 : Bool;
   轴10原点 AT %M1419.6 : Bool;
   轴10到达 AT %M1419.7 : Bool;
   轴11定位1手动 AT %M1420.0 : Bool;
   轴11定位2手动 AT %M1420.1 : Bool;
   轴11定位3手动 AT %M1420.2 : Bool;
   轴11定位4手动 AT %M1420.3 : Bool;
   轴11xx1手动 AT %M1420.4 : Bool;
   轴11xx2手动 AT %M1420.5 : Bool;
   轴11xx3手动 AT %M1420.6 : Bool;
   轴11xx4手动 AT %M1420.7 : Bool;
   轴11使能 AT %M1421.0 : Bool;
   轴11回零 AT %M1421.1 : Bool;
   "轴11点动+" AT %M1421.2 : Bool;
   "轴11点动-" AT %M1421.3 : Bool;
   轴11自由定位 AT %M1421.4 : Bool;
   轴11就绪 AT %M1421.5 : Bool;
   轴11原点 AT %M1421.6 : Bool;
   轴11到达 AT %M1421.7 : Bool;
   轴12定位1手动 AT %M1422.0 : Bool;
   轴12定位2手动 AT %M1422.1 : Bool;
   轴12定位3手动 AT %M1422.2 : Bool;
   轴12定位4手动 AT %M1422.3 : Bool;
   轴12xx1手动 AT %M1422.4 : Bool;
   轴12xx2手动 AT %M1422.5 : Bool;
   轴12xx3手动 AT %M1422.6 : Bool;
   轴12xx4手动 AT %M1422.7 : Bool;
   轴12使能 AT %M1423.0 : Bool;
   轴12回零 AT %M1423.1 : Bool;
   "轴12点动+" AT %M1423.2 : Bool;
   "轴12点动-" AT %M1423.3 : Bool;
   轴12自由定位 AT %M1423.4 : Bool;
   轴12就绪 AT %M1423.5 : Bool;
   轴12原点 AT %M1423.6 : Bool;
   轴12到达 AT %M1423.7 : Bool;
   轴13定位1手动 AT %M1424.0 : Bool;
   轴13定位2手动 AT %M1424.1 : Bool;
   轴13定位3手动 AT %M1424.2 : Bool;
   轴13定位4手动 AT %M1424.3 : Bool;
   轴13xx1手动 AT %M1424.4 : Bool;
   轴13xx2手动 AT %M1424.5 : Bool;
   轴13xx3手动 AT %M1424.6 : Bool;
   轴13xx4手动 AT %M1424.7 : Bool;
   轴13使能 AT %M1425.0 : Bool;
   轴13回零 AT %M1425.1 : Bool;
   "轴13点动+" AT %M1425.2 : Bool;
   "轴13点动-" AT %M1425.3 : Bool;
   轴13自由定位 AT %M1425.4 : Bool;
   轴13就绪 AT %M1425.5 : Bool;
   轴13原点 AT %M1425.6 : Bool;
   轴13到达 AT %M1425.7 : Bool;
   轴14定位1手动 AT %M1426.0 : Bool;
   轴14定位2手动 AT %M1426.1 : Bool;
   轴14定位3手动 AT %M1426.2 : Bool;
   轴14定位4手动 AT %M1426.3 : Bool;
   轴14xx1手动 AT %M1426.4 : Bool;
   轴14xx2手动 AT %M1426.5 : Bool;
   轴14xx3手动 AT %M1426.6 : Bool;
   轴14xx4手动 AT %M1426.7 : Bool;
   轴14使能 AT %M1427.0 : Bool;
   轴14回零 AT %M1427.1 : Bool;
   "轴14点动+" AT %M1427.2 : Bool;
   "轴14点动-" AT %M1427.3 : Bool;
   轴14自由定位 AT %M1427.4 : Bool;
   轴14就绪 AT %M1427.5 : Bool;
   轴14原点 AT %M1427.6 : Bool;
   轴14到达 AT %M1427.7 : Bool;
   轴15定位1手动 AT %M1428.0 : Bool;
   轴15定位2手动 AT %M1428.1 : Bool;
   轴15定位3手动 AT %M1428.2 : Bool;
   轴15定位4手动 AT %M1428.3 : Bool;
   轴15xx1手动 AT %M1428.4 : Bool;
   轴15xx2手动 AT %M1428.5 : Bool;
   轴15xx3手动 AT %M1428.6 : Bool;
   轴15xx4手动 AT %M1428.7 : Bool;
   轴15使能 AT %M1429.0 : Bool;
   轴15回零 AT %M1429.1 : Bool;
   "轴15点动+" AT %M1429.2 : Bool;
   "轴15点动-" AT %M1429.3 : Bool;
   轴15自由定位 AT %M1429.4 : Bool;
   轴15就绪 AT %M1429.5 : Bool;
   轴15原点 AT %M1429.6 : Bool;
   轴15到达 AT %M1429.7 : Bool;
   轴16定位1手动 AT %M1430.0 : Bool;
   轴16定位2手动 AT %M1430.1 : Bool;
   轴16定位3手动 AT %M1430.2 : Bool;
   轴16定位4手动 AT %M1430.3 : Bool;
   轴16xx1手动 AT %M1430.4 : Bool;
   轴16xx2手动 AT %M1430.5 : Bool;
   轴16xx3手动 AT %M1430.6 : Bool;
   轴16xx4手动 AT %M1430.7 : Bool;
   轴16使能 AT %M1431.0 : Bool;
   轴16回零 AT %M1431.1 : Bool;
   "轴16点动+" AT %M1431.2 : Bool;
   "轴16点动-" AT %M1431.3 : Bool;
   轴16自由定位 AT %M1431.4 : Bool;
   轴16就绪 AT %M1431.5 : Bool;
   轴16原点 AT %M1431.6 : Bool;
   轴16到达 AT %M1431.7 : Bool;
   XXXXXX2 AT %M1432.0 : Bool;
   轴1定位1到位 AT %M3400.0 : Bool;
   轴1定位2到位 AT %M3400.1 : Bool;
   轴1定位3到位 AT %M3400.2 : Bool;
   轴1定位4到位 AT %M3400.3 : Bool;
   轴2定位1到位 AT %M3401.0 : Bool;
   轴2定位2到位 AT %M3401.1 : Bool;
   轴2定位3到位 AT %M3401.2 : Bool;
   轴2定位4到位 AT %M3401.3 : Bool;
   轴3定位1到位 AT %M3402.0 : Bool;
   轴3定位2到位 AT %M3402.1 : Bool;
   轴3定位3到位 AT %M3402.2 : Bool;
   轴3定位4到位 AT %M3402.3 : Bool;
   轴4定位1到位 AT %M3403.0 : Bool;
   轴4定位2到位 AT %M3403.1 : Bool;
   轴4定位3到位 AT %M3403.2 : Bool;
   轴4定位4到位 AT %M3403.3 : Bool;
   轴5定位1到位 AT %M3404.0 : Bool;
   轴5定位2到位 AT %M3404.1 : Bool;
   轴5定位3到位 AT %M3404.2 : Bool;
   轴5定位4到位 AT %M3404.3 : Bool;
   轴6定位1到位 AT %M3405.0 : Bool;
   轴6定位2到位 AT %M3405.1 : Bool;
   轴6定位3到位 AT %M3405.2 : Bool;
   轴6定位4到位 AT %M3405.3 : Bool;
   轴7定位1到位 AT %M3406.0 : Bool;
   轴7定位2到位 AT %M3406.1 : Bool;
   轴7定位3到位 AT %M3406.2 : Bool;
   轴7定位4到位 AT %M3406.3 : Bool;
   轴8定位1到位 AT %M3407.0 : Bool;
   轴8定位2到位 AT %M3407.1 : Bool;
   轴8定位3到位 AT %M3407.2 : Bool;
   轴8定位4到位 AT %M3407.3 : Bool;
   轴9定位1到位 AT %M3408.0 : Bool;
   轴9定位2到位 AT %M3408.1 : Bool;
   轴9定位3到位 AT %M3408.2 : Bool;
   轴9定位4到位 AT %M3408.3 : Bool;
   轴10定位1到位 AT %M3409.0 : Bool;
   轴10定位2到位 AT %M3409.1 : Bool;
   轴10定位3到位 AT %M3409.2 : Bool;
   轴10定位4到位 AT %M3409.3 : Bool;
   轴11定位1到位 AT %M3410.0 : Bool;
   轴11定位2到位 AT %M3410.1 : Bool;
   轴11定位3到位 AT %M3410.2 : Bool;
   轴11定位4到位 AT %M3410.3 : Bool;
   轴12定位1到位 AT %M3411.0 : Bool;
   轴12定位2到位 AT %M3411.1 : Bool;
   轴12定位3到位 AT %M3411.2 : Bool;
   轴12定位4到位 AT %M3411.3 : Bool;
   轴13定位1到位 AT %M3412.0 : Bool;
   轴13定位2到位 AT %M3412.1 : Bool;
   轴13定位3到位 AT %M3412.2 : Bool;
   轴13定位4到位 AT %M3412.3 : Bool;
   轴14定位1到位 AT %M3413.0 : Bool;
   轴14定位2到位 AT %M3413.1 : Bool;
   轴14定位3到位 AT %M3413.2 : Bool;
   轴14定位4到位 AT %M3413.3 : Bool;
   轴15定位1到位 AT %M3414.0 : Bool;
   轴15定位2到位 AT %M3414.1 : Bool;
   轴15定位3到位 AT %M3414.2 : Bool;
   轴15定位4到位 AT %M3414.3 : Bool;
   轴16定位1到位 AT %M3415.0 : Bool;
   轴16定位2到位 AT %M3415.1 : Bool;
   轴16定位3到位 AT %M3415.2 : Bool;
   轴16定位4到位 AT %M3415.3 : Bool;
   XXXXXX3 AT %M3416.0 : Bool;
   轴1回零高速 AT %MD1500 : DInt;
   轴1回零低速 AT %MD1504 : DInt;
   轴1点动速度 AT %MD1508 : DInt;
   轴1最高速度 AT %MD1512 : DInt;
   轴1自由定位值 AT %MD1516 : DInt;
   轴2回零高速 AT %MD1520 : DInt;
   轴2回零低速 AT %MD1524 : DInt;
   轴2点动速度 AT %MD1528 : DInt;
   轴2最高速度 AT %MD1532 : DInt;
   轴2自由定位值 AT %MD1536 : DInt;
   轴3回零高速 AT %MD1540 : DInt;
   轴3回零低速 AT %MD1544 : DInt;
   轴3点动速度 AT %MD1548 : DInt;
   轴3最高速度 AT %MD1552 : DInt;
   轴3自由定位值 AT %MD1556 : DInt;
   轴4回零高速 AT %MD1560 : DInt;
   轴4回零低速 AT %MD1564 : DInt;
   轴4点动速度 AT %MD1568 : DInt;
   轴4最高速度 AT %MD1572 : DInt;
   轴4自由定位值 AT %MD1576 : DInt;
   轴5回零高速 AT %MD1580 : DInt;
   轴5回零低速 AT %MD1584 : DInt;
   轴5点动速度 AT %MD1588 : DInt;
   轴5最高速度 AT %MD1592 : DInt;
   轴5自由定位值 AT %MD1596 : DInt;
   轴6回零高速 AT %MD1600 : DInt;
   轴6回零低速 AT %MD1604 : DInt;
   轴6点动速度 AT %MD1608 : DInt;
   轴6最高速度 AT %MD1612 : DInt;
   轴6自由定位值 AT %MD1616 : DInt;
   轴7回零高速 AT %MD1620 : DInt;
   轴7回零低速 AT %MD1624 : DInt;
   轴7点动速度 AT %MD1628 : DInt;
   轴7最高速度 AT %MD1632 : DInt;
   轴7自由定位值 AT %MD1636 : DInt;
   轴8回零高速 AT %MD1640 : DInt;
   轴8回零低速 AT %MD1644 : DInt;
   轴8点动速度 AT %MD1648 : DInt;
   轴8最高速度 AT %MD1652 : DInt;
   轴8自由定位值 AT %MD1656 : DInt;
   轴9回零高速 AT %MD1660 : DInt;
   轴9回零低速 AT %MD1664 : DInt;
   轴9点动速度 AT %MD1668 : DInt;
   轴9最高速度 AT %MD1672 : DInt;
   轴9自由定位值 AT %MD1676 : DInt;
   轴10回零高速 AT %MD1680 : DInt;
   轴10回零低速 AT %MD1684 : DInt;
   轴10点动速度 AT %MD1688 : DInt;
   轴10最高速度 AT %MD1692 : DInt;
   轴10自由定位值 AT %MD1696 : DInt;
   轴11回零高速 AT %MD1700 : DInt;
   轴11回零低速 AT %MD1704 : DInt;
   轴11点动速度 AT %MD1708 : DInt;
   轴11最高速度 AT %MD1712 : DInt;
   轴11自由定位值 AT %MD1716 : DInt;
   轴12回零高速 AT %MD1720 : DInt;
   轴12回零低速 AT %MD1724 : DInt;
   轴12点动速度 AT %MD1728 : DInt;
   轴12最高速度 AT %MD1732 : DInt;
   轴12自由定位值 AT %MD1736 : DInt;
   轴13回零高速 AT %MD1740 : DInt;
   轴13回零低速 AT %MD1744 : DInt;
   轴13点动速度 AT %MD1748 : DInt;
   轴13最高速度 AT %MD1752 : DInt;
   轴13自由定位值 AT %MD1756 : DInt;
   轴14回零高速 AT %MD1760 : DInt;
   轴14回零低速 AT %MD1764 : DInt;
   轴14点动速度 AT %MD1768 : DInt;
   轴14最高速度 AT %MD1772 : DInt;
   轴14自由定位值 AT %MD1776 : DInt;
   轴15回零高速 AT %MD1780 : DInt;
   轴15回零低速 AT %MD1784 : DInt;
   轴15点动速度 AT %MD1788 : DInt;
   轴15最高速度 AT %MD1792 : DInt;
   轴15自由定位值 AT %MD1796 : DInt;
   轴16回零高速 AT %MD1800 : DInt;
   轴16回零低速 AT %MD1804 : DInt;
   轴16点动速度 AT %MD1808 : DInt;
   轴16最高速度 AT %MD1812 : DInt;
   轴16自由定位值 AT %MD1816 : DInt;
   XXXXXX4 AT %MW1920 : Int;
   轴1位置1 AT %MD2500 : DInt;
   轴1位置2 AT %MD2504 : DInt;
   轴1位置3 AT %MD2508 : DInt;
   轴1位置4 AT %MD2512 : DInt;
   轴2位置1 AT %MD2520 : DInt;
   轴2位置2 AT %MD2524 : DInt;
   轴2位置3 AT %MD2528 : DInt;
   轴2位置4 AT %MD2532 : DInt;
   轴3位置1 AT %MD2540 : DInt;
   轴3位置2 AT %MD2544 : DInt;
   轴3位置3 AT %MD2548 : DInt;
   轴3位置4 AT %MD2552 : DInt;
   轴4位置1 AT %MD2560 : DInt;
   轴4位置2 AT %MD2564 : DInt;
   轴4位置3 AT %MD2568 : DInt;
   轴4位置4 AT %MD2572 : DInt;
   轴5位置1 AT %MD2580 : DInt;
   轴5位置2 AT %MD2584 : DInt;
   轴5位置3 AT %MD2588 : DInt;
   轴5位置4 AT %MD2592 : DInt;
   轴6位置1 AT %MD2600 : DInt;
   轴6位置2 AT %MD2604 : DInt;
   轴6位置3 AT %MD2608 : DInt;
   轴6位置4 AT %MD2612 : DInt;
   轴7位置1 AT %MD2620 : DInt;
   轴7位置2 AT %MD2624 : DInt;
   轴7位置3 AT %MD2628 : DInt;
   轴7位置4 AT %MD2632 : DInt;
   轴8位置1 AT %MD2640 : DInt;
   轴8位置2 AT %MD2644 : DInt;
   轴8位置3 AT %MD2648 : DInt;
   轴8位置4 AT %MD2652 : DInt;
   轴9位置1 AT %MD2660 : DInt;
   轴9位置2 AT %MD2664 : DInt;
   轴9位置3 AT %MD2668 : DInt;
   轴9位置4 AT %MD2672 : DInt;
   轴10位置1 AT %MD2680 : DInt;
   轴10位置2 AT %MD2684 : DInt;
   轴10位置3 AT %MD2688 : DInt;
   轴10位置4 AT %MD2692 : DInt;
   轴11位置1 AT %MD2700 : DInt;
   轴11位置2 AT %MD2704 : DInt;
   轴11位置3 AT %MD2708 : DInt;
   轴11位置4 AT %MD2712 : DInt;
   轴12位置1 AT %MD2720 : DInt;
   轴12位置2 AT %MD2724 : DInt;
   轴12位置3 AT %MD2728 : DInt;
   轴12位置4 AT %MD2732 : DInt;
   轴13位置1 AT %MD2740 : DInt;
   轴13位置2 AT %MD2744 : DInt;
   轴13位置3 AT %MD2748 : DInt;
   轴13位置4 AT %MD2752 : DInt;
   轴14位置1 AT %MD2760 : DInt;
   轴14位置2 AT %MD2764 : DInt;
   轴14位置3 AT %MD2768 : DInt;
   轴14位置4 AT %MD2772 : DInt;
   轴15位置1 AT %MD2780 : DInt;
   轴15位置2 AT %MD2784 : DInt;
   轴15位置3 AT %MD2788 : DInt;
   轴15位置4 AT %MD2792 : DInt;
   轴16位置1 AT %MD2800 : DInt;
   轴16位置2 AT %MD2804 : DInt;
   轴16位置3 AT %MD2808 : DInt;
   轴16位置4 AT %MD2812 : DInt;
   XXXXXX5 AT %MW2820 : Int;
   轴1速度1 AT %MW3500 : Int;
   轴1速度2 AT %MW3504 : Int;
   轴1速度3 AT %MW3508 : Int;
   轴1速度4 AT %MW3512 : Int;
   轴2速度1 AT %MW3520 : Int;
   轴2速度2 AT %MW3524 : Int;
   轴2速度3 AT %MW3528 : Int;
   轴2速度4 AT %MW3532 : Int;
   轴3速度1 AT %MW3540 : Int;
   轴3速度2 AT %MW3544 : Int;
   轴3速度3 AT %MW3548 : Int;
   轴3速度4 AT %MW3552 : Int;
   轴4速度1 AT %MW3560 : Int;
   轴4速度2 AT %MW3564 : Int;
   轴4速度3 AT %MW3568 : Int;
   轴4速度4 AT %MW3572 : Int;
   轴5速度1 AT %MW3580 : Int;
   轴5速度2 AT %MW3584 : Int;
   轴5速度3 AT %MW3588 : Int;
   轴5速度4 AT %MW3592 : Int;
   轴6速度1 AT %MW3600 : Int;
   轴6速度2 AT %MW3604 : Int;
   轴6速度3 AT %MW3608 : Int;
   轴6速度4 AT %MW3612 : Int;
   轴7速度1 AT %MW3620 : Int;
   轴7速度2 AT %MW3624 : Int;
   轴7速度3 AT %MW3628 : Int;
   轴7速度4 AT %MW3632 : Int;
   轴8速度1 AT %MW3640 : Int;
   轴8速度2 AT %MW3644 : Int;
   轴8速度3 AT %MW3648 : Int;
   轴8速度4 AT %MW3652 : Int;
   轴9速度1 AT %MW3660 : Int;
   轴9速度2 AT %MW3664 : Int;
   轴9速度3 AT %MW3668 : Int;
   轴9速度4 AT %MW3672 : Int;
   轴10速度1 AT %MW3680 : Int;
   轴10速度2 AT %MW3684 : Int;
   轴10速度3 AT %MW3688 : Int;
   轴10速度4 AT %MW3692 : Int;
   轴11速度1 AT %MW3700 : Int;
   轴11速度2 AT %MW3704 : Int;
   轴11速度3 AT %MW3708 : Int;
   轴11速度4 AT %MW3712 : Int;
   轴12速度1 AT %MW3720 : Int;
   轴12速度2 AT %MW3724 : Int;
   轴12速度3 AT %MW3728 : Int;
   轴12速度4 AT %MW3732 : Int;
   轴13速度1 AT %MW3740 : Int;
   轴13速度2 AT %MW3744 : Int;
   轴13速度3 AT %MW3748 : Int;
   轴13速度4 AT %MW3752 : Int;
   轴14速度1 AT %MW3760 : Int;
   轴14速度2 AT %MW3764 : Int;
   轴14速度3 AT %MW3768 : Int;
   轴14速度4 AT %MW3772 : Int;
   轴15速度1 AT %MW3780 : Int;
   轴15速度2 AT %MW3784 : Int;
   轴15速度3 AT %MW3788 : Int;
   轴15速度4 AT %MW3792 : Int;
   轴16速度1 AT %MW3800 : Int;
   轴16速度2 AT %MW3804 : Int;
   轴16速度3 AT %MW3808 : Int;
   轴16速度4 AT %MW3812 : Int;
   XXXXXX6 AT %MW3820 : Int;
   轴01目标位置 AT %MD4500 : DInt;
   轴02目标位置 AT %MD4504 : DInt;
   轴03目标位置 AT %MD4508 : DInt;
   轴04目标位置 AT %MD4512 : DInt;
   轴05目标位置 AT %MD4516 : DInt;
   轴06目标位置 AT %MD4520 : DInt;
   轴07目标位置 AT %MD4524 : DInt;
   轴08目标位置 AT %MD4528 : DInt;
   轴09目标位置 AT %MD4532 : DInt;
   轴10目标位置 AT %MD4536 : DInt;
   轴11目标位置 AT %MD4540 : DInt;
   轴12目标位置 AT %MD4544 : DInt;
   轴13目标位置 AT %MD4548 : DInt;
   轴14目标位置 AT %MD4552 : DInt;
   轴15目标位置 AT %MD4556 : DInt;
   轴16目标位置 AT %MD4560 : DInt;
   XXXXXX7 AT %MD4564 : DInt;
   轴01目标速度 AT %MD4600 : DInt;
   轴02目标速度 AT %MD4604 : DInt;
   轴03目标速度 AT %MD4608 : DInt;
   轴04目标速度 AT %MD4612 : DInt;
   轴05目标速度 AT %MD4616 : DInt;
   轴06目标速度 AT %MD4620 : DInt;
   轴07目标速度 AT %MD4624 : DInt;
   轴08目标速度 AT %MD4628 : DInt;
   轴09目标速度 AT %MD4632 : DInt;
   轴10目标速度 AT %MD4636 : DInt;
   轴11目标速度 AT %MD4640 : DInt;
   轴12目标速度 AT %MD4644 : DInt;
   轴13目标速度 AT %MD4648 : DInt;
   轴14目标速度 AT %MD4652 : DInt;
   轴15目标速度 AT %MD4656 : DInt;
   轴16目标速度 AT %MD4660 : DInt;
   XXXXXX8 AT %MD4664 : DInt;
   轴01当前位置 AT %MD4700 : DInt;
   轴02当前位置 AT %MD4704 : DInt;
   轴03当前位置 AT %MD4708 : DInt;
   轴04当前位置 AT %MD4712 : DInt;
   轴05当前位置 AT %MD4716 : DInt;
   轴06当前位置 AT %MD4720 : DInt;
   轴07当前位置 AT %MD4724 : DInt;
   轴08当前位置 AT %MD4728 : DInt;
   轴09当前位置 AT %MD4732 : DInt;
   轴10当前位置 AT %MD4736 : DInt;
   轴11当前位置 AT %MD4740 : DInt;
   轴12当前位置 AT %MD4744 : DInt;
   轴13当前位置 AT %MD4748 : DInt;
   轴14当前位置 AT %MD4752 : DInt;
   轴15当前位置 AT %MD4756 : DInt;
   轴16当前位置 AT %MD4760 : DInt;
   XXXXXX9 AT %MD4764 : DInt;
   轴01当前速度 AT %MD4800 : DInt;
   轴02当前速度 AT %MD4804 : DInt;
   轴03当前速度 AT %MD4808 : DInt;
   轴04当前速度 AT %MD4812 : DInt;
   轴05当前速度 AT %MD4816 : DInt;
   轴06当前速度 AT %MD4820 : DInt;
   轴07当前速度 AT %MD4824 : DInt;
   轴08当前速度 AT %MD4828 : DInt;
   轴09当前速度 AT %MD4832 : DInt;
   轴10当前速度 AT %MD4836 : DInt;
   轴11当前速度 AT %MD4840 : DInt;
   轴12当前速度 AT %MD4844 : DInt;
   轴13当前速度 AT %MD4848 : DInt;
   轴14当前速度 AT %MD4852 : DInt;
   轴15当前速度 AT %MD4856 : DInt;
   轴16当前速度 AT %MD4860 : DInt;
   XXXXXX10 AT %MD4864 : DInt;
   轴1报警码 AT %MW4900 : Word;
   轴2报警码 AT %MW4901 : Word;
   轴3报警码 AT %MW4902 : Word;
   轴4报警码 AT %MW4903 : Word;
   轴5报警码 AT %MW4904 : Word;
   轴6报警码 AT %MW4905 : Word;
   轴7报警码 AT %MW4906 : Word;
   轴8报警码 AT %MW4907 : Word;
   轴9报警码 AT %MW4908 : Word;
   轴10报警码 AT %MW4909 : Word;
   轴11报警码 AT %MW4910 : Word;
   轴12报警码 AT %MW4911 : Word;
   轴13报警码 AT %MW4912 : Word;
   轴14报警码 AT %MW4913 : Word;
   轴15报警码 AT %MW4914 : Word;
   轴16报警码 AT %MW4915 : Word;
   XXXXXX11 AT %MW4916 : Word;
   轴1错误码 AT %MW4920 : Word;
   轴2错误码 AT %MW4921 : Word;
   轴3错误码 AT %MW4922 : Word;
   轴4错误码 AT %MW4923 : Word;
   轴5错误码 AT %MW4924 : Word;
   轴6错误码 AT %MW4925 : Word;
   轴7错误码 AT %MW4926 : Word;
   轴8错误码 AT %MW4927 : Word;
   轴9错误码 AT %MW4928 : Word;
   轴10错误码 AT %MW4929 : Word;
   轴11错误码 AT %MW4930 : Word;
   轴12错误码 AT %MW4931 : Word;
   轴13错误码 AT %MW4932 : Word;
   轴14错误码 AT %MW4933 : Word;
   轴15错误码 AT %MW4934 : Word;
   轴16错误码 AT %MW4935 : Word;
END_VAR

DATA_BLOCK "00_WCS交互"   // DB1000
{ S7_Optimized_Access := 'TRUE' }
VERSION : 0.1
// stored: AutoNumber false, DBAccessibleFromOPCUA true, IsOnlyStoredInLoadMemory false, IsRetainMemResEnabled false, IsWriteProtectedInAS false, MemoryReserve 100
BEGIN
END_DATA_BLOCK

DATA_BLOCK "10_前工序交互"   // DB1010
{ S7_Optimized_Access := 'TRUE' }
VERSION : 0.1
// stored: AutoNumber false, DBAccessibleFromOPCUA true, IsOnlyStoredInLoadMemory false, IsRetainMemResEnabled false, IsWriteProtectedInAS false, MemoryReserve 100
BEGIN
END_DATA_BLOCK

DATA_BLOCK "20_后工序交互"   // DB1020
{ S7_Optimized_Access := 'TRUE' }
VERSION : 0.1
// stored: AutoNumber false, DBAccessibleFromOPCUA true, IsOnlyStoredInLoadMemory false, IsRetainMemResEnabled false, IsWriteProtectedInAS false, MemoryReserve 100
BEGIN
END_DATA_BLOCK

DATA_BLOCK "Com_DB"   // DB1
{ S7_Optimized_Access := 'TRUE' }
VERSION : 0.1
// stored: AutoNumber false, DBAccessibleFromOPCUA true, IsOnlyStoredInLoadMemory false, IsRetainMemResEnabled false, IsWriteProtectedInAS false, MemoryReserve 0
   VAR
      K01 : Struct   // S01使用
         "M" : Bool;
      END_STRUCT;
      K02 : Struct
         ST1_InitCont : Bool;   // ST1初始化条件
         ST1_InitStart : Bool;   // ST1初始化启动
      END_STRUCT;
      K03 : Struct
         InitTon2S { S7_SetPoint := 'True'} : IEC_TIMER;   // 初始2S
         PlcRunTon2s { S7_SetPoint := 'True'} : IEC_TIMER;   // 运行2秒
         PlcRunTon3s { S7_SetPoint := 'True'} : IEC_TIMER;   // 运行3秒
         PlcRunTon4s { S7_SetPoint := 'True'} : IEC_TIMER;   // 运行4秒
         EN_托盘在席 : Bool;
         EN_托盘离席 : Bool;
         EN_前端LS_ON { S7_SetPoint := 'True'} : IEC_TIMER;
         EN_前端LS_OFF { S7_SetPoint := 'True'} : IEC_TIMER;
         EN_后端LS_ON { S7_SetPoint := 'True'} : IEC_TIMER;
         EN_后端LS_OFF { S7_SetPoint := 'True'} : IEC_TIMER;
         EX_托盘在席 : Bool;
         EX_托盘离席 : Bool;
         EX_前端LS_ON { S7_SetPoint := 'True'} : IEC_TIMER;
         EX_前端LS_OFF { S7_SetPoint := 'True'} : IEC_TIMER;
         EX_后端LS_ON { S7_SetPoint := 'True'} : IEC_TIMER;
         EX_后端LS_OFF { S7_SetPoint := 'True'} : IEC_TIMER;
         ST01上托盘在席 : Bool;
         ST01上托盘离席 : Bool;
         ST01上前端LS_ON { S7_SetPoint := 'True'} : IEC_TIMER;
         ST01上前端LS_OFF { S7_SetPoint := 'True'} : IEC_TIMER;
         ST01上后端LS_ON { S7_SetPoint := 'True'} : IEC_TIMER;
         ST01上后端LS_OFF { S7_SetPoint := 'True'} : IEC_TIMER;
         ST01下托盘在席 : Bool;
         ST01下托盘离席 : Bool;
         ST01下前端LS_ON { S7_SetPoint := 'True'} : IEC_TIMER;
         ST01下前端LS_OFF { S7_SetPoint := 'True'} : IEC_TIMER;
         ST01下后端LS_ON { S7_SetPoint := 'True'} : IEC_TIMER;
         ST01下后端LS_OFF { S7_SetPoint := 'True'} : IEC_TIMER;
         ST02上托盘在席 : Bool;
         ST02上托盘离席 : Bool;
         ST02上前端LS_ON { S7_SetPoint := 'True'} : IEC_TIMER;
         ST02上前端LS_OFF { S7_SetPoint := 'True'} : IEC_TIMER;
         ST02上后端LS_ON { S7_SetPoint := 'True'} : IEC_TIMER;
         ST02上后端LS_OFF { S7_SetPoint := 'True'} : IEC_TIMER;
         ST02下托盘在席 : Bool;
         ST02下托盘离席 : Bool;
         ST02下前端LS_ON { S7_SetPoint := 'True'} : IEC_TIMER;
         ST02下前端LS_OFF { S7_SetPoint := 'True'} : IEC_TIMER;
         ST02下后端LS_ON { S7_SetPoint := 'True'} : IEC_TIMER;
         ST02下后端LS_OFF { S7_SetPoint := 'True'} : IEC_TIMER;
         ST03上托盘在席 : Bool;
         ST03上托盘离席 : Bool;
         ST03上前端LS_ON { S7_SetPoint := 'True'} : IEC_TIMER;
         ST03上前端LS_OFF { S7_SetPoint := 'True'} : IEC_TIMER;
         ST03上后端LS_ON { S7_SetPoint := 'True'} : IEC_TIMER;
         ST03上后端LS_OFF { S7_SetPoint := 'True'} : IEC_TIMER;
         ST03下托盘在席 : Bool;
         ST03下托盘离席 : Bool;
         ST03下前端LS_ON { S7_SetPoint := 'True'} : IEC_TIMER;
         ST03下前端LS_OFF { S7_SetPoint := 'True'} : IEC_TIMER;
         ST03下后端LS_ON { S7_SetPoint := 'True'} : IEC_TIMER;
         ST03下后端LS_OFF { S7_SetPoint := 'True'} : IEC_TIMER;
         ST04上托盘在席 : Bool;
         ST04上托盘离席 : Bool;
         ST04上前端LS_ON { S7_SetPoint := 'True'} : IEC_TIMER;
         ST04上前端LS_OFF { S7_SetPoint := 'True'} : IEC_TIMER;
         ST04上后端LS_ON { S7_SetPoint := 'True'} : IEC_TIMER;
         ST04上后端LS_OFF { S7_SetPoint := 'True'} : IEC_TIMER;
         ST05上托盘在席 : Bool;
         ST05上托盘离席 : Bool;
         ST05上前端LS_ON { S7_SetPoint := 'True'} : IEC_TIMER;
         ST05上前端LS_OFF { S7_SetPoint := 'True'} : IEC_TIMER;
         ST05上后端LS_ON { S7_SetPoint := 'True'} : IEC_TIMER;
         ST05上后端LS_OFF { S7_SetPoint := 'True'} : IEC_TIMER;
         ST06上托盘在席 : Bool;
         ST06上托盘离席 : Bool;
         ST06上前端LS_ON { S7_SetPoint := 'True'} : IEC_TIMER;
         ST06上前端LS_OFF { S7_SetPoint := 'True'} : IEC_TIMER;
         ST06上后端LS_ON { S7_SetPoint := 'True'} : IEC_TIMER;
         ST06上后端LS_OFF { S7_SetPoint := 'True'} : IEC_TIMER;
         ST07上托盘在席 : Bool;
         ST07上托盘离席 : Bool;
         ST07上前端LS_ON { S7_SetPoint := 'True'} : IEC_TIMER;
         ST07上前端LS_OFF { S7_SetPoint := 'True'} : IEC_TIMER;
         ST07上后端LS_ON { S7_SetPoint := 'True'} : IEC_TIMER;
         ST07上后端LS_OFF { S7_SetPoint := 'True'} : IEC_TIMER;
         ST08上托盘在席 : Bool;
         ST08上托盘离席 : Bool;
         ST08上前端LS_ON { S7_SetPoint := 'True'} : IEC_TIMER;
         ST08上前端LS_OFF { S7_SetPoint := 'True'} : IEC_TIMER;
         ST08上后端LS_ON { S7_SetPoint := 'True'} : IEC_TIMER;
         ST08上后端LS_OFF { S7_SetPoint := 'True'} : IEC_TIMER;
         ST09上托盘在席 : Bool;
         ST09上托盘离席 : Bool;
         ST09上前端LS_ON { S7_SetPoint := 'True'} : IEC_TIMER;
         ST09上前端LS_OFF { S7_SetPoint := 'True'} : IEC_TIMER;
         ST09上后端LS_ON { S7_SetPoint := 'True'} : IEC_TIMER;
         ST09上后端LS_OFF { S7_SetPoint := 'True'} : IEC_TIMER;
         ST10上托盘在席 : Bool;
         ST10上托盘离席 : Bool;
         ST10上前端LS_ON { S7_SetPoint := 'True'} : IEC_TIMER;
         ST10上前端LS_OFF { S7_SetPoint := 'True'} : IEC_TIMER;
         ST10上后端LS_ON { S7_SetPoint := 'True'} : IEC_TIMER;
         ST10上后端LS_OFF { S7_SetPoint := 'True'} : IEC_TIMER;
         ST11上托盘在席 : Bool;
         ST11上托盘离席 : Bool;
         ST11上前端LS_ON { S7_SetPoint := 'True'} : IEC_TIMER;
         ST11上前端LS_OFF { S7_SetPoint := 'True'} : IEC_TIMER;
         ST11上后端LS_ON { S7_SetPoint := 'True'} : IEC_TIMER;
         ST11上后端LS_OFF { S7_SetPoint := 'True'} : IEC_TIMER;
         ST12上托盘在席 : Bool;
         ST12上托盘离席 : Bool;
         ST12上前端LS_ON { S7_SetPoint := 'True'} : IEC_TIMER;
         ST12上前端LS_OFF { S7_SetPoint := 'True'} : IEC_TIMER;
         ST12上后端LS_ON { S7_SetPoint := 'True'} : IEC_TIMER;
         ST12上后端LS_OFF { S7_SetPoint := 'True'} : IEC_TIMER;
         ST01按压延迟 { S7_SetPoint := 'True'} : IEC_TIMER;
         ST02按压延迟 { S7_SetPoint := 'True'} : IEC_TIMER;
         ST03按压延迟 { S7_SetPoint := 'True'} : IEC_TIMER;
         ST04按压延迟 { S7_SetPoint := 'True'} : IEC_TIMER;
         ST05按压延迟 { S7_SetPoint := 'True'} : IEC_TIMER;
         ST06按压延迟 { S7_SetPoint := 'True'} : IEC_TIMER;
         ST07按压延迟 { S7_SetPoint := 'True'} : IEC_TIMER;
         ST08按压延迟 { S7_SetPoint := 'True'} : IEC_TIMER;
         ST09按压延迟 { S7_SetPoint := 'True'} : IEC_TIMER;
         ST10按压延迟 { S7_SetPoint := 'True'} : IEC_TIMER;
         ST11按压延迟 { S7_SetPoint := 'True'} : IEC_TIMER;
         ST12按压延迟 { S7_SetPoint := 'True'} : IEC_TIMER;
      END_STRUCT;
      K04 : Struct
         EMO : Array[1..16] of Bool;   // 急停报警
         SLC : Array[1..16] of Bool;   // 光栅报警
         DSW : Array[1..16] of Bool;   // 门SW报警
         OtherSafe : Array[1..16] of Bool;   // 其它安全报警
         AirALM : Array[1..16] of Bool;   // 气压报警
         AirALMTon : Array[1..16] of IEC_TIMER;   // 气压报警延迟
         DrumALM : Array[1..48] of Bool;   // 滚筒报警
         DrumTiOver : Array[1..48] of Bool;   // 滚筒超时
         DrumOverTon : Array[1..48] of IEC_TIMER;   // 滚筒超时延迟
         SensALM : Array[1..48] of Bool;   // 传感器故障
         SensTiOver : Array[1..48] of IEC_TIMER;   // 传感器故障延迟
         MoveALM : Array[1..48] of Bool;   // 动作异常
         MoveALMTiOver : Array[1..48] of IEC_TIMER;   // 动作异常延迟
         InvALM : Array[1..16] of Bool;   // 变频器故障
         InvNoRun : Array[1..16] of Bool;   // 变频器未运行故障
         InvNoRunTon : Array[1..16] of IEC_TIMER;   // 变频器未运行延迟
         InvTiOver : Array[1..16] of Bool;   // 变频器超时故障
         InvOverTon : Array[1..16] of IEC_TIMER;   // 变频器超时延迟
         InvOverload : Array[1..16] of Bool;   // 变频器过负载
         ValAdvTiOver : Array[1..48] of Bool;   // 阀出动作超时
         ValRetTiOver : Array[1..48] of Bool;   // 阀回动作超时
         ValSensALM : Array[1..48] of Bool;   // 阀到位传感器都ON故障
         ValSenCroALM : Array[1..48] of Bool;   // 阀到位传感器交叉ON故障
         AxisWarn : Array[1..16] of Bool;   // 轴警告
         AxisALM : Array[1..16] of Bool;   // 轴故障
         AxisNoReady : Array[1..16] of Bool;   // 轴未准备好
         AxisHomeALM : Array[1..16] of Bool;   // 轴未回零
         AxisNoRun : Array[1..16] of Bool;   // 轴未运行
         AxisNoRunTon : Array[1..16] of IEC_TIMER;   // 轴未运行超时
         AxisFLS : Array[1..16] of Bool;   // 轴正极限
         AxisRLS : Array[1..16] of Bool;   // 轴负极限
         RobotALM : Array[1..16] of Bool;   // 机器人故障
         CCDALM : Array[1..16] of Bool;   // 视觉故障
         CommALM : Array[1..16] of Bool;   // 通信故障
         AnalogUpALM : Array[1..16] of Bool;   // 模拟量上限故障
         AnalogLowALM : Array[1..16] of Bool;   // 模拟量下限故障
         OtherALM : Array[1..16] of Bool;   // 其它故障
      END_STRUCT;
      K05 : Struct
         ManTon { S7_SetPoint := 'True'} : IEC_TIMER;   // 手动延迟
         AutoTon { S7_SetPoint := 'True'} : IEC_TIMER;   // 自动延迟
      END_STRUCT;
      K06 : Struct
         AdvCond_Val { ExternalAccessible := 'False'; ExternalVisible := 'False'; ExternalWritable := 'False'} : Array[1..48] of Bool;   // 阀前进条件
         RetCond_Val { ExternalAccessible := 'False'; ExternalVisible := 'False'; ExternalWritable := 'False'} : Array[1..48] of Bool;   // 阀返回条件
         AdvCond_Drum { ExternalAccessible := 'False'; ExternalVisible := 'False'; ExternalWritable := 'False'} : Array[1..48] of Bool;   // 滚筒正转条件
         RetCond_Drum { ExternalAccessible := 'False'; ExternalVisible := 'False'; ExternalWritable := 'False'} : Array[1..48] of Bool;   // 滚筒反转条件
         AdvCond_Inv : Array[1..16] of Bool;   // 变频器正转条件
         RetCond_Inv : Array[1..16] of Bool;   // 变频器反转条件
      END_STRUCT;
      K07 : Struct
         Axis1Cont : Array[1..8] of Bool;   // 轴1动作条件
         Axis1Start : Bool;   // 轴1定位启动
         Axis1Pulse : Array[1..20] of Bool;   // 轴1脉冲
         Axis1Rate : Array[1..3] of Int;   // 轴1速率
         Axis1TON : Array[1..2] of IEC_TIMER;   // 轴1计时
         Axis2Cont : Array[1..8] of Bool;   // 轴2动作条件
         Axis2Start : Bool;   // 轴2定位启动
         Axis2Pulse : Array[1..20] of Bool;   // 轴2脉冲
         Axis2Rate : Array[1..3] of Int;   // 轴2速率
         Axis2TON : Array[1..2] of IEC_TIMER;   // 轴2计时
         Axis3Cont : Array[1..8] of Bool;   // 轴3动作条件
         Axis3Start : Bool;   // 轴3定位启动
         Axis3Pulse : Array[1..20] of Bool;   // 轴3脉冲
         Axis3Rate : Array[1..3] of Int;   // 轴3速率
         Axis3TON : Array[1..2] of IEC_TIMER;   // 轴3计时
         Axis4Cont : Array[1..8] of Bool;   // 轴4动作条件
         Axis4Start : Bool;   // 轴4定位启动
         Axis4Pulse : Array[1..20] of Bool;   // 轴4脉冲
         Axis4Rate : Array[1..3] of Int;   // 轴4速率
         Axis4TON : Array[1..2] of IEC_TIMER;   // 轴4计时
         Axis5Cont : Array[1..8] of Bool;   // 轴5动作条件
         Axis5Start : Bool;   // 轴5定位启动
         Axis5Pulse : Array[1..20] of Bool;   // 轴5脉冲
         Axis5Rate : Array[1..3] of Int;   // 轴5速率
         Axis5TON : Array[1..2] of IEC_TIMER;   // 轴5计时
         Axis6Cont : Array[1..8] of Bool;   // 轴6动作条件
         Axis6Start : Bool;   // 轴6定位启动
         Axis6Pulse : Array[1..20] of Bool;   // 轴6脉冲
         Axis6Rate : Array[1..3] of Int;   // 轴6速率
         Axis6TON : Array[1..2] of IEC_TIMER;   // 轴6计时
         Axis7Cont : Array[1..8] of Bool;   // 轴7动作条件
         Axis7Start : Bool;   // 轴7定位启动
         Axis7Pulse : Array[1..20] of Bool;   // 轴7脉冲
         Axis7Rate : Array[1..3] of Int;   // 轴7速率
         Axis7TON : Array[1..2] of IEC_TIMER;   // 轴7计时
         Axis8Cont : Array[1..8] of Bool;   // 轴8动作条件
         Axis8Start : Bool;   // 轴8定位启动
         Axis8Pulse : Array[1..20] of Bool;   // 轴8脉冲
         Axis8Rate : Array[1..3] of Int;   // 轴8速率
         Axis8TON : Array[1..2] of IEC_TIMER;   // 轴8计时
         Axis9Cont : Array[1..8] of Bool;   // 轴9动作条件
         Axis9Start : Bool;   // 轴9定位启动
         Axis9Pulse : Array[1..20] of Bool;   // 轴9脉冲
         Axis9Rate : Array[1..3] of Int;   // 轴9速率
         Axis9TON : Array[1..2] of IEC_TIMER;   // 轴9计时
         Axis10Cont : Array[1..8] of Bool;   // 轴10动作条件
         Axis10Start : Bool;   // 轴10定位启动
         Axis10Pulse : Array[1..20] of Bool;   // 轴10脉冲
         Axis10Rate : Array[1..3] of Int;   // 轴10速率
         Axis10TON : Array[1..2] of IEC_TIMER;   // 轴10计时
         Axis11Cont : Array[1..8] of Bool;   // 轴11动作条件
         Axis11Start : Bool;   // 轴11定位启动
         Axis11Pulse : Array[1..20] of Bool;   // 轴11脉冲
         Axis11Rate : Array[1..3] of Int;   // 轴11速率
         Axis11TON : Array[1..2] of IEC_TIMER;   // 轴11计时
         Axis12Cont : Array[1..8] of Bool;   // 轴12动作条件
         Axis12Start : Bool;   // 轴12定位启动
         Axis12Pulse : Array[1..20] of Bool;   // 轴12脉冲
         Axis12Rate : Array[1..3] of Int;   // 轴12速率
         Axis12TON : Array[1..2] of IEC_TIMER;   // 轴12计时
         Axis13Cont : Array[1..8] of Bool;   // 轴13动作条件
         Axis13Start : Bool;   // 轴13定位启动
         Axis13Pulse : Array[1..20] of Bool;   // 轴13脉冲
         Axis13Rate : Array[1..3] of Int;   // 轴13速率
         Axis13TON : Array[1..2] of IEC_TIMER;   // 轴13计时
         Axis14Cont : Array[1..8] of Bool;   // 轴14动作条件
         Axis14Start : Bool;   // 轴14定位启动
         Axis14Pulse : Array[1..20] of Bool;   // 轴4脉冲
         Axis14Rate : Array[1..3] of Int;   // 轴14速率
         Axis14TON : Array[1..2] of IEC_TIMER;   // 轴14计时
         Axis15Cont : Array[1..8] of Bool;   // 轴15动作条件
         Axis15Start : Bool;   // 轴15定位启动
         Axis15Pulse : Array[1..20] of Bool;   // 轴15脉冲
         Axis15Rate : Array[1..3] of Int;   // 轴15速率
         Axis15TON : Array[1..2] of IEC_TIMER;   // 轴15计时
         Axis16Cont : Array[1..8] of Bool;   // 轴16动作条件
         Axis16Start : Bool;   // 轴16定位启动
         Axis16Pulse : Array[1..20] of Bool;   // 轴16脉冲
         Axis16Rate : Array[1..3] of Int;   // 轴16速率
         Axis16TON : Array[1..2] of IEC_TIMER;   // 轴16计时
      END_STRUCT;
      K08 : Struct
         "M" : Bool;   // 位
      END_STRUCT;
      K10 : Struct
         "M" : Bool;   // 位
      END_STRUCT;
      K40 : Struct
         "M" : Bool;   // 位
      END_STRUCT;
   END_VAR
BEGIN
   // K04.ValAdvTiOver[1] : 阀1出动作超时
   // K04.ValAdvTiOver[2] : 阀2出动作超时
   // K04.ValAdvTiOver[3] : 阀3出动作超时
   // K04.ValAdvTiOver[4] : 阀4出动作超时
   // K04.ValAdvTiOver[5] : 阀5出动作超时
   // K04.ValAdvTiOver[6] : 阀6出动作超时
   // K04.ValAdvTiOver[7] : 阀7出动作超时
   // K04.ValAdvTiOver[8] : 阀8出动作超时
   // K04.ValRetTiOver[1] : 阀1回动作超时
   // K04.ValRetTiOver[2] : 阀2回动作超时
   // K04.ValRetTiOver[3] : 阀3回动作超时
   // K04.ValRetTiOver[4] : 阀4回动作超时
   // K04.ValRetTiOver[5] : 阀5回动作超时
   // K04.ValRetTiOver[6] : 阀6回动作超时
   // K04.ValRetTiOver[7] : 阀7回动作超时
   // K04.ValRetTiOver[8] : 阀8回动作超时
   // K06.AdvCond_Val[1] : 阀1前进条件
   // K06.AdvCond_Val[2] : 阀2前进条件
   // K06.AdvCond_Val[3] : 阀3前进条件
   // K06.AdvCond_Val[4] : 阀4前进条件
   // K06.AdvCond_Val[5] : 阀5前进条件
   // K06.AdvCond_Val[6] : 阀6前进条件
   // K06.AdvCond_Val[7] : 阀7前进条件
   // K06.AdvCond_Val[8] : 阀8前进条件
   // K06.AdvCond_Val[9] : 阀9前进条件
   // K06.AdvCond_Val[10] : 阀10前进条件
   // K06.AdvCond_Val[11] : 阀11前进条件
   // K06.AdvCond_Val[12] : 阀12前进条件
   // K06.AdvCond_Val[13] : 阀13前进条件
   // K06.AdvCond_Val[14] : 阀14前进条件
   // K06.AdvCond_Val[15] : 阀15前进条件
   // K06.AdvCond_Val[16] : 阀16前进条件
   // K06.AdvCond_Val[17] : 阀17前进条件
   // K06.AdvCond_Val[18] : 阀18前进条件
   // K06.AdvCond_Val[19] : 阀19前进条件
   // K06.AdvCond_Val[20] : 阀20前进条件
   // K06.AdvCond_Val[21] : 阀21前进条件
   // K06.AdvCond_Val[22] : 阀22前进条件
   // K06.AdvCond_Val[23] : 阀23前进条件
   // K06.AdvCond_Val[24] : 阀24前进条件
   // K06.AdvCond_Val[25] : 阀25前进条件
   // K06.AdvCond_Val[26] : 阀26前进条件
   // K06.AdvCond_Val[27] : 阀27前进条件
   // K06.AdvCond_Val[28] : 阀28前进条件
   // K06.AdvCond_Val[29] : 阀29前进条件
   // K06.AdvCond_Val[30] : 阀30前进条件
   // K06.AdvCond_Val[31] : 阀31前进条件
   // K06.AdvCond_Val[32] : 阀32前进条件
   // K06.AdvCond_Val[33] : 阀33前进条件
   // K06.AdvCond_Val[34] : 阀34前进条件
   // K06.AdvCond_Val[35] : 阀35前进条件
   // K06.AdvCond_Val[36] : 阀36前进条件
   // K06.AdvCond_Val[37] : 阀37前进条件
   // K06.AdvCond_Val[38] : 阀38前进条件
   // K06.AdvCond_Val[39] : 阀39前进条件
   // K06.AdvCond_Val[40] : 阀40前进条件
   // K06.AdvCond_Val[41] : 阀41前进条件
   // K06.AdvCond_Val[42] : 阀42前进条件
   // K06.AdvCond_Val[43] : 阀43前进条件
   // K06.AdvCond_Val[44] : 阀44前进条件
   // K06.AdvCond_Val[45] : 阀45前进条件
   // K06.AdvCond_Val[46] : 阀46前进条件
   // K06.AdvCond_Val[47] : 阀47前进条件
   // K06.AdvCond_Val[48] : 阀48前进条件
   // K06.RetCond_Val[1] : 阀1返回条件
   // K06.RetCond_Val[2] : 阀2返回条件
   // K06.RetCond_Val[3] : 阀3返回条件
   // K06.RetCond_Val[4] : 阀4返回条件
   // K06.RetCond_Val[5] : 阀5返回条件
   // K06.RetCond_Val[6] : 阀6返回条件
   // K06.RetCond_Val[7] : 阀7返回条件
   // K06.RetCond_Val[8] : 阀8返回条件
   // K06.RetCond_Val[9] : 阀9返回条件
   // K06.RetCond_Val[10] : 阀10返回条件
   // K06.RetCond_Val[11] : 阀11返回条件
   // K06.RetCond_Val[12] : 阀12返回条件
   // K06.RetCond_Val[13] : 阀13返回条件
   // K06.RetCond_Val[14] : 阀14返回条件
   // K06.RetCond_Val[15] : 阀15返回条件
   // K06.RetCond_Val[16] : 阀16返回条件
   // K06.RetCond_Val[17] : 阀17返回条件
   // K06.RetCond_Val[18] : 阀18返回条件
   // K06.RetCond_Val[19] : 阀19返回条件
   // K06.RetCond_Val[20] : 阀20返回条件
   // K06.RetCond_Val[21] : 阀21返回条件
   // K06.RetCond_Val[22] : 阀22返回条件
   // K06.RetCond_Val[23] : 阀23返回条件
   // K06.RetCond_Val[24] : 阀24返回条件
   // K06.RetCond_Val[25] : 阀25返回条件
   // K06.RetCond_Val[26] : 阀26返回条件
   // K06.RetCond_Val[27] : 阀27返回条件
   // K06.RetCond_Val[28] : 阀28返回条件
   // K06.RetCond_Val[29] : 阀29返回条件
   // K06.RetCond_Val[30] : 阀30返回条件
   // K06.RetCond_Val[31] : 阀31返回条件
   // K06.RetCond_Val[32] : 阀32返回条件
   // K06.RetCond_Val[33] : 阀33返回条件
   // K06.RetCond_Val[34] : 阀34返回条件
   // K06.RetCond_Val[35] : 阀35返回条件
   // K06.RetCond_Val[36] : 阀36返回条件
   // K06.RetCond_Val[37] : 阀37返回条件
   // K06.RetCond_Val[38] : 阀38返回条件
   // K06.RetCond_Val[39] : 阀39返回条件
   // K06.RetCond_Val[40] : 阀40返回条件
   // K06.RetCond_Val[41] : 阀41返回条件
   // K06.RetCond_Val[42] : 阀42返回条件
   // K06.RetCond_Val[43] : 阀43返回条件
   // K06.RetCond_Val[44] : 阀44返回条件
   // K06.RetCond_Val[45] : 阀45返回条件
   // K06.RetCond_Val[46] : 阀46返回条件
   // K06.RetCond_Val[47] : 阀47返回条件
   // K06.RetCond_Val[48] : 阀48返回条件
   // K07.Axis1Cont[1] : 共同条件
   // K07.Axis1Cont[2] : 回零条件
   // K07.Axis1Cont[3] : JOG正条件
   // K07.Axis1Cont[4] : JOG负条件
   // K07.Axis1Cont[5] : 定位正条件
   // K07.Axis1Cont[6] : 定位负条件
   // K07.Axis1Cont[7] : 预留
   // K07.Axis1Cont[8] : 预留
   // K07.Axis1Rate[1] : 轴1速率%
   // K07.Axis1Rate[2] : 轴1加速速率%
   // K07.Axis1Rate[3] : 轴1减速速率%
   // K07.Axis2Cont[1] : 共同条件
   // K07.Axis2Cont[2] : 回零条件
   // K07.Axis2Cont[3] : JOG正条件
   // K07.Axis2Cont[4] : JOG负条件
   // K07.Axis2Cont[5] : 定位正条件
   // K07.Axis2Cont[6] : 定位负条件
   // K07.Axis2Cont[7] : 预留
   // K07.Axis2Cont[8] : 预留
   // K07.Axis2Rate[1] : 轴1速率%
   // K07.Axis2Rate[2] : 轴1加速速率%
   // K07.Axis2Rate[3] : 轴1减速速率%
   // K07.Axis3Cont[1] : 共同条件
   // K07.Axis3Cont[2] : 回零条件
   // K07.Axis3Cont[3] : JOG正条件
   // K07.Axis3Cont[4] : JOG负条件
   // K07.Axis3Cont[5] : 定位正条件
   // K07.Axis3Cont[6] : 定位负条件
   // K07.Axis3Cont[7] : 预留
   // K07.Axis3Cont[8] : 预留
   // K07.Axis3Rate[1] : 轴1速率%
   // K07.Axis3Rate[2] : 轴1加速速率%
   // K07.Axis3Rate[3] : 轴1减速速率%
   // K07.Axis4Cont[1] : 共同条件
   // K07.Axis4Cont[2] : 回零条件
   // K07.Axis4Cont[3] : JOG正条件
   // K07.Axis4Cont[4] : JOG负条件
   // K07.Axis4Cont[5] : 定位正条件
   // K07.Axis4Cont[6] : 定位负条件
   // K07.Axis4Cont[7] : 预留
   // K07.Axis4Cont[8] : 预留
   // K07.Axis4Rate[1] : 轴1速率%
   // K07.Axis4Rate[2] : 轴1加速速率%
   // K07.Axis4Rate[3] : 轴1减速速率%
   // K07.Axis5Cont[1] : 共同条件
   // K07.Axis5Cont[2] : 回零条件
   // K07.Axis5Cont[3] : JOG正条件
   // K07.Axis5Cont[4] : JOG负条件
   // K07.Axis5Cont[5] : 定位正条件
   // K07.Axis5Cont[6] : 定位负条件
   // K07.Axis5Cont[7] : 预留
   // K07.Axis5Cont[8] : 预留
   // K07.Axis5Rate[1] : 轴1速率%
   // K07.Axis5Rate[2] : 轴1加速速率%
   // K07.Axis5Rate[3] : 轴1减速速率%
   // K07.Axis6Cont[1] : 共同条件
   // K07.Axis6Cont[2] : 回零条件
   // K07.Axis6Cont[3] : JOG正条件
   // K07.Axis6Cont[4] : JOG负条件
   // K07.Axis6Cont[5] : 定位正条件
   // K07.Axis6Cont[6] : 定位负条件
   // K07.Axis6Cont[7] : 预留
   // K07.Axis6Cont[8] : 预留
   // K07.Axis6Rate[1] : 轴1速率%
   // K07.Axis6Rate[2] : 轴1加速速率%
   // K07.Axis6Rate[3] : 轴1减速速率%
   // K07.Axis7Cont[1] : 共同条件
   // K07.Axis7Cont[2] : 回零条件
   // K07.Axis7Cont[3] : JOG正条件
   // K07.Axis7Cont[4] : JOG负条件
   // K07.Axis7Cont[5] : 定位正条件
   // K07.Axis7Cont[6] : 定位负条件
   // K07.Axis7Cont[7] : 预留
   // K07.Axis7Cont[8] : 预留
   // K07.Axis7Rate[1] : 轴1速率%
   // K07.Axis7Rate[2] : 轴1加速速率%
   // K07.Axis7Rate[3] : 轴1减速速率%
   // K07.Axis8Cont[1] : 共同条件
   // K07.Axis8Cont[2] : 回零条件
   // K07.Axis8Cont[3] : JOG正条件
   // K07.Axis8Cont[4] : JOG负条件
   // K07.Axis8Cont[5] : 定位正条件
   // K07.Axis8Cont[6] : 定位负条件
   // K07.Axis8Cont[7] : 预留
   // K07.Axis8Cont[8] : 预留
   // K07.Axis8Rate[1] : 轴1速率%
   // K07.Axis8Rate[2] : 轴1加速速率%
   // K07.Axis8Rate[3] : 轴1减速速率%
   // K07.Axis9Cont[1] : 共同条件
   // K07.Axis9Cont[2] : 回零条件
   // K07.Axis9Cont[3] : JOG正条件
   // K07.Axis9Cont[4] : JOG负条件
   // K07.Axis9Cont[5] : 定位正条件
   // K07.Axis9Cont[6] : 定位负条件
   // K07.Axis9Cont[7] : 预留
   // K07.Axis9Cont[8] : 预留
   // K07.Axis9Rate[1] : 轴1速率%
   // K07.Axis9Rate[2] : 轴1加速速率%
   // K07.Axis9Rate[3] : 轴1减速速率%
   // K07.Axis10Cont[1] : 共同条件
   // K07.Axis10Cont[2] : 回零条件
   // K07.Axis10Cont[3] : JOG正条件
   // K07.Axis10Cont[4] : JOG负条件
   // K07.Axis10Cont[5] : 定位正条件
   // K07.Axis10Cont[6] : 定位负条件
   // K07.Axis10Cont[7] : 预留
   // K07.Axis10Cont[8] : 预留
   // K07.Axis10Rate[1] : 轴1速率%
   // K07.Axis10Rate[2] : 轴1加速速率%
   // K07.Axis10Rate[3] : 轴1减速速率%
   // K07.Axis11Cont[1] : 共同条件
   // K07.Axis11Cont[2] : 回零条件
   // K07.Axis11Cont[3] : JOG正条件
   // K07.Axis11Cont[4] : JOG负条件
   // K07.Axis11Cont[5] : 定位正条件
   // K07.Axis11Cont[6] : 定位负条件
   // K07.Axis11Cont[7] : 预留
   // K07.Axis11Cont[8] : 预留
   // K07.Axis11Rate[1] : 轴1速率%
   // K07.Axis11Rate[2] : 轴1加速速率%
   // K07.Axis11Rate[3] : 轴1减速速率%
   // K07.Axis12Cont[1] : 共同条件
   // K07.Axis12Cont[2] : 回零条件
   // K07.Axis12Cont[3] : JOG正条件
   // K07.Axis12Cont[4] : JOG负条件
   // K07.Axis12Cont[5] : 定位正条件
   // K07.Axis12Cont[6] : 定位负条件
   // K07.Axis12Cont[7] : 预留
   // K07.Axis12Cont[8] : 预留
   // K07.Axis12Rate[1] : 轴1速率%
   // K07.Axis12Rate[2] : 轴1加速速率%
   // K07.Axis12Rate[3] : 轴1减速速率%
   // K07.Axis13Cont[1] : 共同条件
   // K07.Axis13Cont[2] : 回零条件
   // K07.Axis13Cont[3] : JOG正条件
   // K07.Axis13Cont[4] : JOG负条件
   // K07.Axis13Cont[5] : 定位正条件
   // K07.Axis13Cont[6] : 定位负条件
   // K07.Axis13Cont[7] : 预留
   // K07.Axis13Cont[8] : 预留
   // K07.Axis13Rate[1] : 轴1速率%
   // K07.Axis13Rate[2] : 轴1加速速率%
   // K07.Axis13Rate[3] : 轴1减速速率%
   // K07.Axis14Cont[1] : 共同条件
   // K07.Axis14Cont[2] : 回零条件
   // K07.Axis14Cont[3] : JOG正条件
   // K07.Axis14Cont[4] : JOG负条件
   // K07.Axis14Cont[5] : 定位正条件
   // K07.Axis14Cont[6] : 定位负条件
   // K07.Axis14Cont[7] : 预留
   // K07.Axis14Cont[8] : 预留
   // K07.Axis14Rate[1] : 轴1速率%
   // K07.Axis14Rate[2] : 轴1加速速率%
   // K07.Axis14Rate[3] : 轴1减速速率%
   // K07.Axis15Cont[1] : 共同条件
   // K07.Axis15Cont[2] : 回零条件
   // K07.Axis15Cont[3] : JOG正条件
   // K07.Axis15Cont[4] : JOG负条件
   // K07.Axis15Cont[5] : 定位正条件
   // K07.Axis15Cont[6] : 定位负条件
   // K07.Axis15Cont[7] : 预留
   // K07.Axis15Cont[8] : 预留
   // K07.Axis15Rate[1] : 轴1速率%
   // K07.Axis15Rate[2] : 轴1加速速率%
   // K07.Axis15Rate[3] : 轴1减速速率%
   // K07.Axis16Cont[1] : 共同条件
   // K07.Axis16Cont[2] : 回零条件
   // K07.Axis16Cont[3] : JOG正条件
   // K07.Axis16Cont[4] : JOG负条件
   // K07.Axis16Cont[5] : 定位正条件
   // K07.Axis16Cont[6] : 定位负条件
   // K07.Axis16Cont[7] : 预留
   // K07.Axis16Cont[8] : 预留
   // K07.Axis16Rate[1] : 轴1速率%
   // K07.Axis16Rate[2] : 轴1加速速率%
   // K07.Axis16Rate[3] : 轴1减速速率%
END_DATA_BLOCK

ORGANIZATION_BLOCK "Main"   // OB1, LAD, ProgramCycle
TITLE = "Main Program Sweep (Cycle)"
{ S7_Optimized_Access := 'TRUE' }
VERSION : 0.1
// stored: AutoNumber true, IsIECCheckEnabled false, SetENOAutomatically false
   VAR_INPUT
      Initial_Call : Bool;   // Initial call of this OB
      Remanence : Bool;   // =True, if remanent data are available
   END_VAR
   VAR_TEMP
      PLC_Date_Read : DTL;
      PLC_DateState_R : Int;
      PLC_Date_Write : DTL;
      PLC_DateState_W : Int;
      M_pulse : Array[1..10] of Bool;
      W_SecCont : Array[1..5] of Int;
   END_VAR
   VAR_TEMP   // added for the SCL form of the ladder/FBD networks
      _w1 : Bool;
      _w2 : Bool;
   END_VAR
BEGIN

REGION Network 1: FB调用
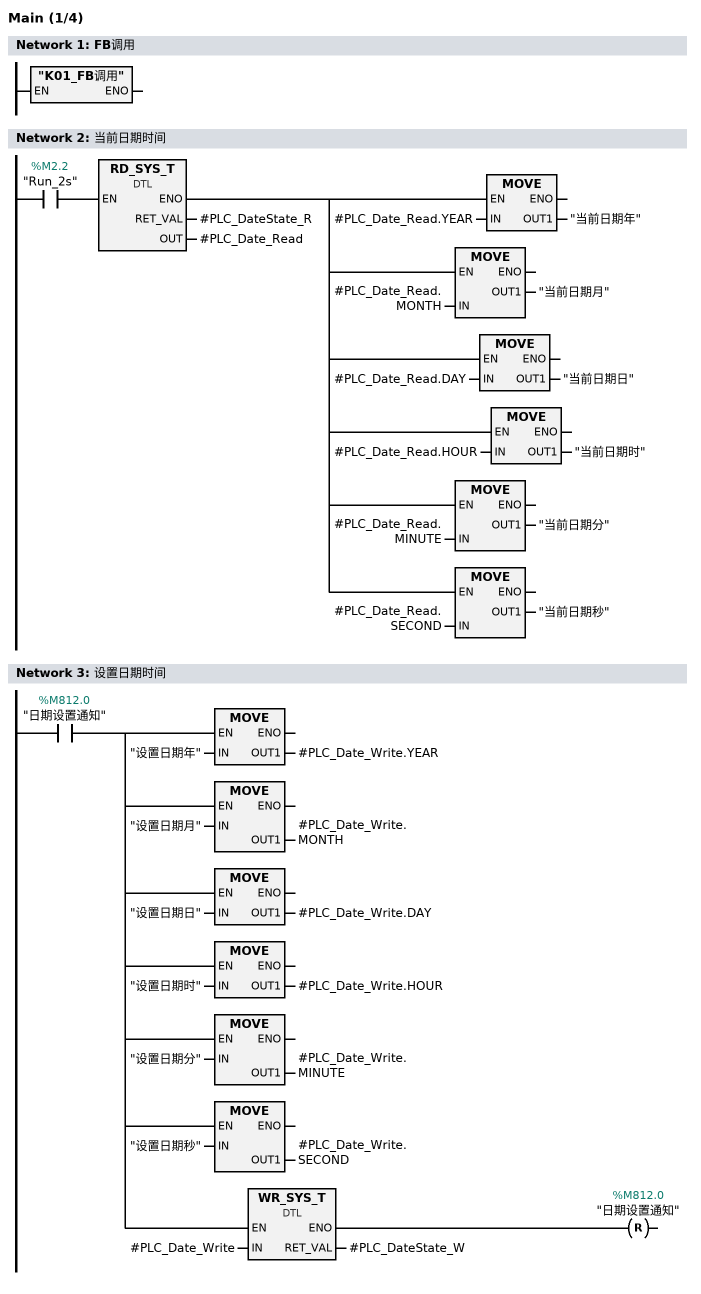
   RUNG wire#powerrail
      "K01_FB调用"()
   END_RUNG
   // the same network as SCL:
   "K01_FB调用"();
END_REGION

REGION Network 2: 当前日期时间
   RUNG wire#powerrail
      Contact( "Run_2s" )
      { S7_Templates := "date_type := DTL" } RD_SYS_T(RET_VAL => #PLC_DateState_R, OUT => #PLC_Date_Read)
      wire#w1
      Move(in := #PLC_Date_Read.YEAR, out1 => "当前日期年")
   END_RUNG
   RUNG wire#w1
      Move(in := #PLC_Date_Read.MONTH, out1 => "当前日期月")
   END_RUNG
   RUNG wire#w1
      Move(in := #PLC_Date_Read.DAY, out1 => "当前日期日")
   END_RUNG
   RUNG wire#w1
      Move(in := #PLC_Date_Read.HOUR, out1 => "当前日期时")
   END_RUNG
   RUNG wire#w1
      Move(in := #PLC_Date_Read.MINUTE, out1 => "当前日期分")
   END_RUNG
   RUNG wire#w1
      Move(in := #PLC_Date_Read.SECOND, out1 => "当前日期秒")
   END_RUNG
   // the same network as SCL:
   #PLC_DateState_R := RD_SYS_T(EN := "Run_2s", OUT => #PLC_Date_Read, ENO => #_w1);
   IF #_w1 THEN
       "当前日期年" := #PLC_Date_Read.YEAR;
       "当前日期月" := #PLC_Date_Read.MONTH;
       "当前日期日" := #PLC_Date_Read.DAY;
       "当前日期时" := #PLC_Date_Read.HOUR;
       "当前日期分" := #PLC_Date_Read.MINUTE;
       "当前日期秒" := #PLC_Date_Read.SECOND;
   END_IF;
END_REGION

REGION Network 3: 设置日期时间
   RUNG wire#powerrail
      Contact( "日期设置通知" )
      wire#w1
      Move(in := "设置日期年", out1 => #PLC_Date_Write.YEAR)
   END_RUNG
   RUNG wire#w1
      Move(in := "设置日期月", out1 => #PLC_Date_Write.MONTH)
   END_RUNG
   RUNG wire#w1
      Move(in := "设置日期日", out1 => #PLC_Date_Write.DAY)
   END_RUNG
   RUNG wire#w1
      Move(in := "设置日期时", out1 => #PLC_Date_Write.HOUR)
   END_RUNG
   RUNG wire#w1
      Move(in := "设置日期分", out1 => #PLC_Date_Write.MINUTE)
   END_RUNG
   RUNG wire#w1
      Move(in := "设置日期秒", out1 => #PLC_Date_Write.SECOND)
   END_RUNG
   RUNG wire#w1
      { S7_Templates := "date_type := DTL" } WR_SYS_T(IN := #PLC_Date_Write, RET_VAL => #PLC_DateState_W)
      R_Coil( "日期设置通知" )
   END_RUNG
   // the same network as SCL:
   IF "日期设置通知" THEN
       #PLC_Date_Write.YEAR := "设置日期年";
       #PLC_Date_Write.MONTH := "设置日期月";
       #PLC_Date_Write.DAY := "设置日期日";
       #PLC_Date_Write.HOUR := "设置日期时";
       #PLC_Date_Write.MINUTE := "设置日期分";
       #PLC_Date_Write.SECOND := "设置日期秒";
   END_IF;
   #PLC_DateState_W := WR_SYS_T(EN := "日期设置通知", IN := #PLC_Date_Write, ENO => #_w1);
   IF #_w1 THEN "日期设置通知" := FALSE; END_IF;
END_REGION

REGION Network 4: 开机日期时间
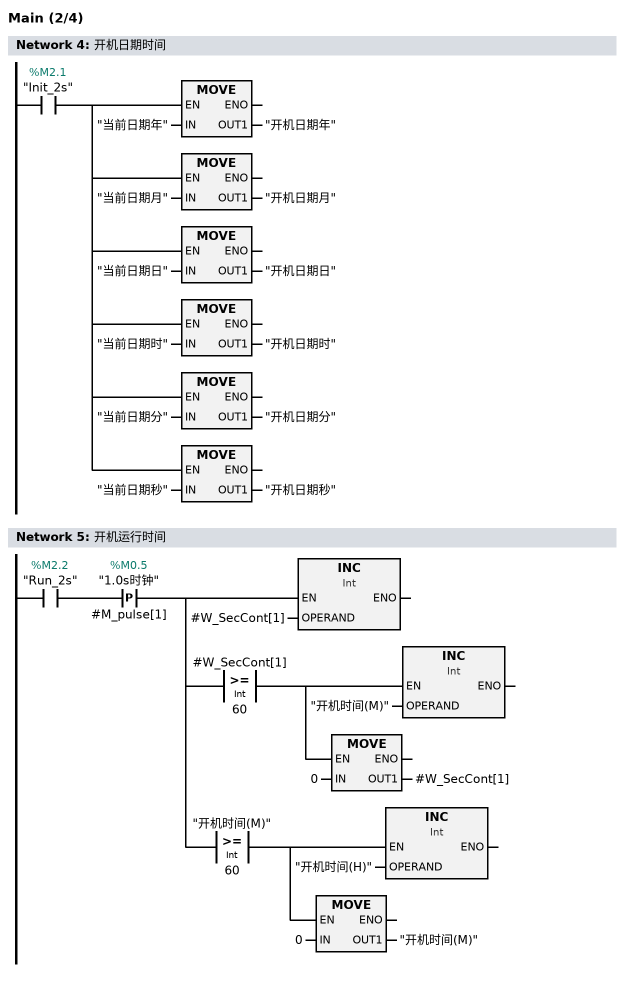
   RUNG wire#powerrail
      Contact( "Init_2s" )
      wire#w1
      Move(in := "当前日期年", out1 => "开机日期年")
   END_RUNG
   RUNG wire#w1
      Move(in := "当前日期月", out1 => "开机日期月")
   END_RUNG
   RUNG wire#w1
      Move(in := "当前日期日", out1 => "开机日期日")
   END_RUNG
   RUNG wire#w1
      Move(in := "当前日期时", out1 => "开机日期时")
   END_RUNG
   RUNG wire#w1
      Move(in := "当前日期分", out1 => "开机日期分")
   END_RUNG
   RUNG wire#w1
      Move(in := "当前日期秒", out1 => "开机日期秒")
   END_RUNG
   // the same network as SCL:
   IF "Init_2s" THEN
       "开机日期年" := "当前日期年";
       "开机日期月" := "当前日期月";
       "开机日期日" := "当前日期日";
       "开机日期时" := "当前日期时";
       "开机日期分" := "当前日期分";
       "开机日期秒" := "当前日期秒";
   END_IF;
END_REGION

REGION Network 5: 开机运行时间
   RUNG wire#powerrail
      Contact( "Run_2s" )
      P_Contact(operand := "1.0s时钟", bit := #M_pulse[1])
      wire#w1
      { S7_Templates := "DestType := Int" } Inc( #W_SecCont[1] )
   END_RUNG
   RUNG wire#w1
      { S7_Templates := "SrcType := Int" } GE_Contact(in1 := #W_SecCont[1], in2 := 60)
      wire#w2
      { S7_Templates := "DestType := Int" } Inc( "开机时间(M)" )
   END_RUNG
   RUNG wire#w2
      Move(in := 0, out1 => #W_SecCont[1])
   END_RUNG
   RUNG wire#w1
      { S7_Templates := "SrcType := Int" } GE_Contact(in1 := "开机时间(M)", in2 := 60)
      wire#w3
      { S7_Templates := "DestType := Int" } Inc( "开机时间(H)" )
   END_RUNG
   RUNG wire#w3
      Move(in := 0, out1 => "开机时间(M)")
   END_RUNG
   // the same network as SCL:
   #_w1 := "Run_2s" AND "1.0s时钟" AND NOT #M_pulse[1];   // rising edge of "1.0s时钟"
   #M_pulse[1] := "1.0s时钟";
   IF #_w1 THEN #W_SecCont[1] := #W_SecCont[1] + 1; END_IF;
   IF #_w1 AND (#W_SecCont[1] >= 60) THEN
       "开机时间(M)" := "开机时间(M)" + 1;
       #W_SecCont[1] := 0;
   END_IF;
   IF #_w1 AND ("开机时间(M)" >= 60) THEN
       "开机时间(H)" := "开机时间(H)" + 1;
       "开机时间(M)" := 0;
   END_IF;
END_REGION

REGION Network 6: 运行时间
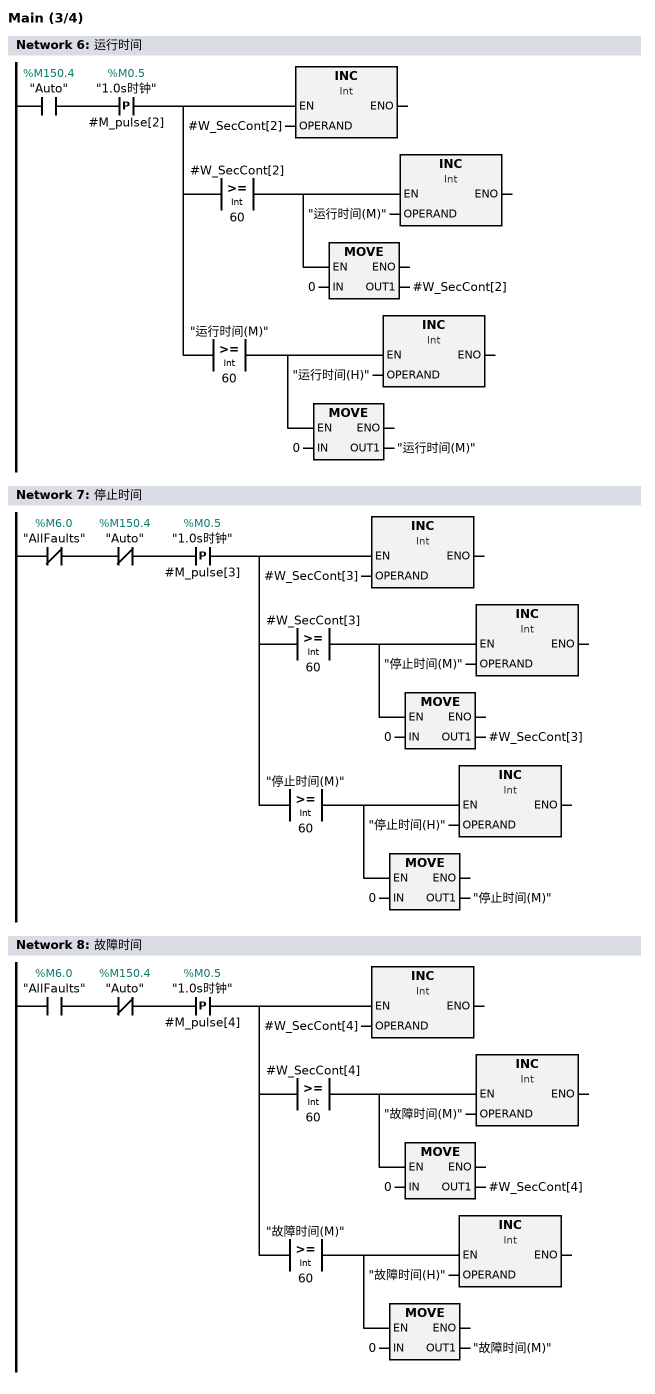
   RUNG wire#powerrail
      Contact( "Auto" )
      P_Contact(operand := "1.0s时钟", bit := #M_pulse[2])
      wire#w1
      { S7_Templates := "DestType := Int" } Inc( #W_SecCont[2] )
   END_RUNG
   RUNG wire#w1
      { S7_Templates := "SrcType := Int" } GE_Contact(in1 := #W_SecCont[2], in2 := 60)
      wire#w2
      { S7_Templates := "DestType := Int" } Inc( "运行时间(M)" )
   END_RUNG
   RUNG wire#w2
      Move(in := 0, out1 => #W_SecCont[2])
   END_RUNG
   RUNG wire#w1
      { S7_Templates := "SrcType := Int" } GE_Contact(in1 := "运行时间(M)", in2 := 60)
      wire#w3
      { S7_Templates := "DestType := Int" } Inc( "运行时间(H)" )
   END_RUNG
   RUNG wire#w3
      Move(in := 0, out1 => "运行时间(M)")
   END_RUNG
   // the same network as SCL:
   #_w1 := "Auto" AND "1.0s时钟" AND NOT #M_pulse[2];   // rising edge of "1.0s时钟"
   #M_pulse[2] := "1.0s时钟";
   IF #_w1 THEN #W_SecCont[2] := #W_SecCont[2] + 1; END_IF;
   IF #_w1 AND (#W_SecCont[2] >= 60) THEN
       "运行时间(M)" := "运行时间(M)" + 1;
       #W_SecCont[2] := 0;
   END_IF;
   IF #_w1 AND ("运行时间(M)" >= 60) THEN
       "运行时间(H)" := "运行时间(H)" + 1;
       "运行时间(M)" := 0;
   END_IF;
END_REGION

REGION Network 7: 停止时间
   RUNG wire#powerrail
      I_Contact( "AllFaults" )
      I_Contact( "Auto" )
      P_Contact(operand := "1.0s时钟", bit := #M_pulse[3])
      wire#w1
      { S7_Templates := "DestType := Int" } Inc( #W_SecCont[3] )
   END_RUNG
   RUNG wire#w1
      { S7_Templates := "SrcType := Int" } GE_Contact(in1 := #W_SecCont[3], in2 := 60)
      wire#w2
      { S7_Templates := "DestType := Int" } Inc( "停止时间(M)" )
   END_RUNG
   RUNG wire#w2
      Move(in := 0, out1 => #W_SecCont[3])
   END_RUNG
   RUNG wire#w1
      { S7_Templates := "SrcType := Int" } GE_Contact(in1 := "停止时间(M)", in2 := 60)
      wire#w3
      { S7_Templates := "DestType := Int" } Inc( "停止时间(H)" )
   END_RUNG
   RUNG wire#w3
      Move(in := 0, out1 => "停止时间(M)")
   END_RUNG
   // the same network as SCL:
   #_w1 := NOT "AllFaults" AND NOT "Auto" AND "1.0s时钟" AND NOT #M_pulse[3];   // rising edge of "1.0s时钟"
   #M_pulse[3] := "1.0s时钟";
   IF #_w1 THEN #W_SecCont[3] := #W_SecCont[3] + 1; END_IF;
   IF #_w1 AND (#W_SecCont[3] >= 60) THEN
       "停止时间(M)" := "停止时间(M)" + 1;
       #W_SecCont[3] := 0;
   END_IF;
   IF #_w1 AND ("停止时间(M)" >= 60) THEN
       "停止时间(H)" := "停止时间(H)" + 1;
       "停止时间(M)" := 0;
   END_IF;
END_REGION

REGION Network 8: 故障时间
   RUNG wire#powerrail
      Contact( "AllFaults" )
      I_Contact( "Auto" )
      P_Contact(operand := "1.0s时钟", bit := #M_pulse[4])
      wire#w1
      { S7_Templates := "DestType := Int" } Inc( #W_SecCont[4] )
   END_RUNG
   RUNG wire#w1
      { S7_Templates := "SrcType := Int" } GE_Contact(in1 := #W_SecCont[4], in2 := 60)
      wire#w2
      { S7_Templates := "DestType := Int" } Inc( "故障时间(M)" )
   END_RUNG
   RUNG wire#w2
      Move(in := 0, out1 => #W_SecCont[4])
   END_RUNG
   RUNG wire#w1
      { S7_Templates := "SrcType := Int" } GE_Contact(in1 := "故障时间(M)", in2 := 60)
      wire#w3
      { S7_Templates := "DestType := Int" } Inc( "故障时间(H)" )
   END_RUNG
   RUNG wire#w3
      Move(in := 0, out1 => "故障时间(M)")
   END_RUNG
   // the same network as SCL:
   #_w1 := "AllFaults" AND NOT "Auto" AND "1.0s时钟" AND NOT #M_pulse[4];   // rising edge of "1.0s时钟"
   #M_pulse[4] := "1.0s时钟";
   IF #_w1 THEN #W_SecCont[4] := #W_SecCont[4] + 1; END_IF;
   IF #_w1 AND (#W_SecCont[4] >= 60) THEN
       "故障时间(M)" := "故障时间(M)" + 1;
       #W_SecCont[4] := 0;
   END_IF;
   IF #_w1 AND ("故障时间(M)" >= 60) THEN
       "故障时间(H)" := "故障时间(H)" + 1;
       "故障时间(M)" := 0;
   END_IF;
END_REGION

REGION Network 9: 实时节拍，工作节拍
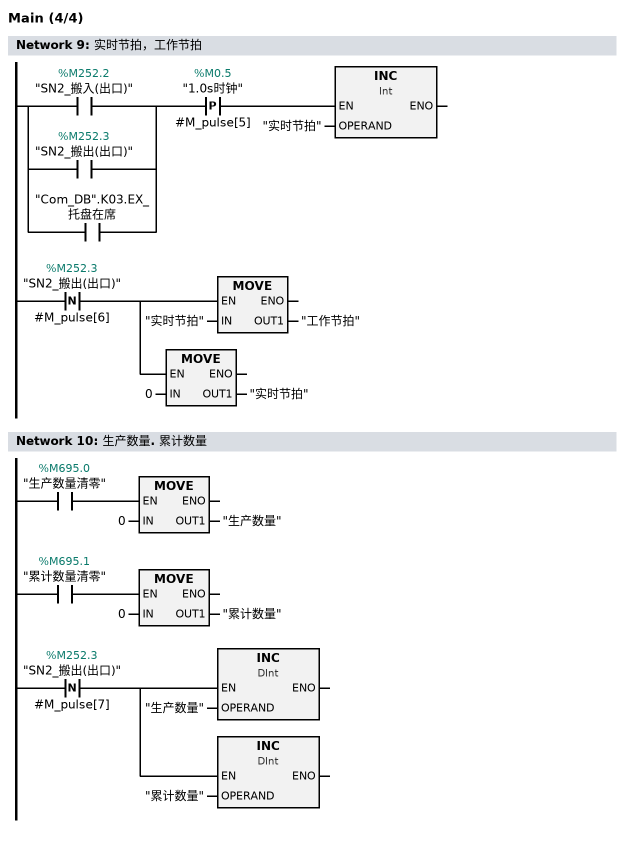
   RUNG wire#powerrail
      Contact( "SN2_搬入(出口)" )
      wire#w1
      P_Contact(operand := "1.0s时钟", bit := #M_pulse[5])
      { S7_Templates := "DestType := Int" } Inc( "实时节拍" )
   END_RUNG
   RUNG wire#powerrail
      Contact( "SN2_搬出(出口)" )
   END_RUNG wire#w1
   RUNG wire#powerrail
      Contact( "Com_DB".K03.EX_托盘在席 )
   END_RUNG wire#w1
   RUNG wire#powerrail
      N_Contact(operand := "SN2_搬出(出口)", bit := #M_pulse[6])
      wire#w2
      Move(in := "实时节拍", out1 => "工作节拍")
   END_RUNG
   RUNG wire#w2
      Move(in := 0, out1 => "实时节拍")
   END_RUNG
   // the same network as SCL:
   #_w1 := ("SN2_搬入(出口)" OR "SN2_搬出(出口)" OR "Com_DB".K03.EX_托盘在席) AND "1.0s时钟" AND NOT #M_pulse[5];   // rising edge of "1.0s时钟"
   #M_pulse[5] := "1.0s时钟";
   IF #_w1 THEN "实时节拍" := "实时节拍" + 1; END_IF;
   #_w2 := NOT "SN2_搬出(出口)" AND #M_pulse[6];   // falling edge of "SN2_搬出(出口)"
   #M_pulse[6] := "SN2_搬出(出口)";
   IF #_w2 THEN
       "工作节拍" := "实时节拍";
       "实时节拍" := 0;
   END_IF;
END_REGION

REGION Network 10: 生产数量. 累计数量
   RUNG wire#powerrail
      Contact( "生产数量清零" )
      Move(in := 0, out1 => "生产数量")
   END_RUNG
   RUNG wire#powerrail
      Contact( "累计数量清零" )
      Move(in := 0, out1 => "累计数量")
   END_RUNG
   RUNG wire#powerrail
      N_Contact(operand := "SN2_搬出(出口)", bit := #M_pulse[7])
      wire#w1
      { S7_Templates := "DestType := DInt" } Inc( "生产数量" )
   END_RUNG
   RUNG wire#w1
      { S7_Templates := "DestType := DInt" } Inc( "累计数量" )
   END_RUNG
   // the same network as SCL:
   IF "生产数量清零" THEN "生产数量" := 0; END_IF;
   IF "累计数量清零" THEN "累计数量" := 0; END_IF;
   #_w1 := NOT "SN2_搬出(出口)" AND #M_pulse[7];   // falling edge of "SN2_搬出(出口)"
   #M_pulse[7] := "SN2_搬出(出口)";
   IF #_w1 THEN
       "生产数量" := "生产数量" + 1;
       "累计数量" := "累计数量" + 1;
   END_IF;
END_REGION

REGION Network 11: OK. NG数量
END_REGION

REGION Network 12 (SCL): 稼动率 合格率 PPM计算

